(* Logix 5000 project; controller reports 1756-L63 rev 20.11; software revision 20.04; part 22 of 52 *)

        [1402].log_data[6].valid := 1, [1402].log_data[7].valid := 1, [1402].log_data[8].valid := 1, [1402].log_data[9].valid := 1, [1402].log_data[10].valid := 1, [1402].log_data[11].valid := 1, [1402].log_data[12].valid := 1, [1402].log_data[13].valid := 1, [1402].log_data[14].valid := 1, [1402].log_data[15].valid := 1, [1402].log_data[16].valid := 1, [1402].log_data[17].valid := 1, [1402].log_data[18].valid := 1, [1402].log_data[19].valid := 1, [1402].time.Year := 2023, [1402].time.Month := 1, [1402].time.Day := 14, [1402].time.Hour := 13, [1402].time.Minute := 14, [1402].time.Second := 59, [1403].log_data[0].min := 1.0, [1403].log_data[0].max := 1.0, [1403].log_data[0].total := 300.0, [1403].log_data[0].time := 300.0, [1403].log_data[0].minminute := 15, [1403].log_data[0].maxminute := 15, [1403].log_data[0].valid := 1, [1403].log_data[1].valid := 1, [1403].log_data[2].valid := 1, [1403].log_data[3].valid := 1, [1403].log_data[4].valid := 1, [1403].log_data[5].valid := 1, [1403].log_data[6].valid := 1, [1403].log_data[7].valid := 1, [1403].log_data[8].valid := 1, [1403].log_data[9].valid := 1, [1403].log_data[10].valid := 1, [1403].log_data[11].valid := 1, [1403].log_data[12].valid := 1, [1403].log_data[13].valid := 1, [1403].log_data[14].valid := 1, [1403].log_data[15].valid := 1, [1403].log_data[16].valid := 1, [1403].log_data[17].valid := 1, [1403].log_data[18].valid := 1, [1403].log_data[19].valid := 1, [1403].time.Year := 2023, [1403].time.Month := 1, [1403].time.Day := 14, [1403].time.Hour := 13, [1403].time.Minute := 19, [1403].time.Second := 59, [1404].log_data[0].min := 1.0, [1404].log_data[0].max := 1.0, [1404].log_data[0].total := 300.0, [1404].log_data[0].time := 300.0, [1404].log_data[0].minminute := 20, [1404].log_data[0].maxminute := 20, [1404].log_data[0].valid := 1, [1404].log_data[1].valid := 1,
        [1404].log_data[2].valid := 1, [1404].log_data[3].valid := 1, [1404].log_data[4].valid := 1, [1404].log_data[5].valid := 1, [1404].log_data[6].valid := 1, [1404].log_data[7].valid := 1, [1404].log_data[8].valid := 1, [1404].log_data[9].valid := 1, [1404].log_data[10].valid := 1, [1404].log_data[11].valid := 1, [1404].log_data[12].valid := 1, [1404].log_data[13].valid := 1, [1404].log_data[14].valid := 1, [1404].log_data[15].valid := 1, [1404].log_data[16].valid := 1, [1404].log_data[17].valid := 1, [1404].log_data[18].valid := 1, [1404].log_data[19].valid := 1, [1404].time.Year := 2023, [1404].time.Month := 1, [1404].time.Day := 14, [1404].time.Hour := 13, [1404].time.Minute := 24, [1404].time.Second := 59, [1405].log_data[0].min := 1.0, [1405].log_data[0].max := 1.0, [1405].log_data[0].total := 300.0, [1405].log_data[0].time := 300.0, [1405].log_data[0].minminute := 25, [1405].log_data[0].maxminute := 25, [1405].log_data[0].valid := 1, [1405].log_data[1].valid := 1, [1405].log_data[2].valid := 1, [1405].log_data[3].valid := 1, [1405].log_data[4].valid := 1, [1405].log_data[5].valid := 1, [1405].log_data[6].valid := 1, [1405].log_data[7].valid := 1, [1405].log_data[8].valid := 1, [1405].log_data[9].valid := 1, [1405].log_data[10].valid := 1, [1405].log_data[11].valid := 1, [1405].log_data[12].valid := 1, [1405].log_data[13].valid := 1, [1405].log_data[14].valid := 1, [1405].log_data[15].valid := 1, [1405].log_data[16].valid := 1, [1405].log_data[17].valid := 1, [1405].log_data[18].valid := 1, [1405].log_data[19].valid := 1, [1405].time.Year := 2023, [1405].time.Month := 1, [1405].time.Day := 14, [1405].time.Hour := 13, [1405].time.Minute := 29, [1405].time.Second := 59, [1406].log_data[0].min := 1.0, [1406].log_data[0].max := 1.0, [1406].log_data[0].total := 300.0, [1406].log_data[0].time := 300.0,
        [1406].log_data[0].minminute := 30, [1406].log_data[0].maxminute := 30, [1406].log_data[0].valid := 1, [1406].log_data[1].valid := 1, [1406].log_data[2].valid := 1, [1406].log_data[3].valid := 1, [1406].log_data[4].valid := 1, [1406].log_data[5].valid := 1, [1406].log_data[6].valid := 1, [1406].log_data[7].valid := 1, [1406].log_data[8].valid := 1, [1406].log_data[9].valid := 1, [1406].log_data[10].valid := 1, [1406].log_data[11].valid := 1, [1406].log_data[12].valid := 1, [1406].log_data[13].valid := 1, [1406].log_data[14].valid := 1, [1406].log_data[15].valid := 1, [1406].log_data[16].valid := 1, [1406].log_data[17].valid := 1, [1406].log_data[18].valid := 1, [1406].log_data[19].valid := 1, [1406].time.Year := 2023, [1406].time.Month := 1, [1406].time.Day := 14, [1406].time.Hour := 13, [1406].time.Minute := 34, [1406].time.Second := 59, [1407].log_data[0].min := 1.0, [1407].log_data[0].max := 1.0, [1407].log_data[0].total := 300.0, [1407].log_data[0].time := 300.0, [1407].log_data[0].minminute := 35, [1407].log_data[0].maxminute := 35, [1407].log_data[0].valid := 1, [1407].log_data[1].valid := 1, [1407].log_data[2].valid := 1, [1407].log_data[3].valid := 1, [1407].log_data[4].valid := 1, [1407].log_data[5].valid := 1, [1407].log_data[6].valid := 1, [1407].log_data[7].valid := 1, [1407].log_data[8].valid := 1, [1407].log_data[9].valid := 1, [1407].log_data[10].valid := 1, [1407].log_data[11].valid := 1, [1407].log_data[12].valid := 1, [1407].log_data[13].valid := 1, [1407].log_data[14].valid := 1, [1407].log_data[15].valid := 1, [1407].log_data[16].valid := 1, [1407].log_data[17].valid := 1, [1407].log_data[18].valid := 1, [1407].log_data[19].valid := 1, [1407].time.Year := 2023, [1407].time.Month := 1, [1407].time.Day := 14, [1407].time.Hour := 13, [1407].time.Minute := 39, [1407].time.Second := 59,
        [1408].log_data[0].min := 1.0, [1408].log_data[0].max := 1.0, [1408].log_data[0].total := 300.0, [1408].log_data[0].time := 300.0, [1408].log_data[0].minminute := 40, [1408].log_data[0].maxminute := 40, [1408].log_data[0].valid := 1, [1408].log_data[1].valid := 1, [1408].log_data[2].valid := 1, [1408].log_data[3].valid := 1, [1408].log_data[4].valid := 1, [1408].log_data[5].valid := 1, [1408].log_data[6].valid := 1, [1408].log_data[7].valid := 1, [1408].log_data[8].valid := 1, [1408].log_data[9].valid := 1, [1408].log_data[10].valid := 1, [1408].log_data[11].valid := 1, [1408].log_data[12].valid := 1, [1408].log_data[13].valid := 1, [1408].log_data[14].valid := 1, [1408].log_data[15].valid := 1, [1408].log_data[16].valid := 1, [1408].log_data[17].valid := 1, [1408].log_data[18].valid := 1, [1408].log_data[19].valid := 1, [1408].time.Year := 2023, [1408].time.Month := 1, [1408].time.Day := 14, [1408].time.Hour := 13, [1408].time.Minute := 44, [1408].time.Second := 59, [1409].log_data[0].min := 1.0, [1409].log_data[0].max := 1.0, [1409].log_data[0].total := 300.0, [1409].log_data[0].time := 300.0, [1409].log_data[0].minminute := 45, [1409].log_data[0].maxminute := 45, [1409].log_data[0].valid := 1, [1409].log_data[1].valid := 1, [1409].log_data[2].valid := 1, [1409].log_data[3].valid := 1, [1409].log_data[4].valid := 1, [1409].log_data[5].valid := 1, [1409].log_data[6].valid := 1, [1409].log_data[7].valid := 1, [1409].log_data[8].valid := 1, [1409].log_data[9].valid := 1, [1409].log_data[10].valid := 1, [1409].log_data[11].valid := 1, [1409].log_data[12].valid := 1, [1409].log_data[13].valid := 1, [1409].log_data[14].valid := 1, [1409].log_data[15].valid := 1, [1409].log_data[16].valid := 1, [1409].log_data[17].valid := 1, [1409].log_data[18].valid := 1, [1409].log_data[19].valid := 1, [1409].time.Year := 2023, [1409].time.Month := 1,
        [1409].time.Day := 14, [1409].time.Hour := 13, [1409].time.Minute := 49, [1409].time.Second := 59, [1410].log_data[0].min := 1.0, [1410].log_data[0].max := 1.0, [1410].log_data[0].total := 300.0, [1410].log_data[0].time := 300.0, [1410].log_data[0].minminute := 50, [1410].log_data[0].maxminute := 50, [1410].log_data[0].valid := 1, [1410].log_data[1].valid := 1, [1410].log_data[2].valid := 1, [1410].log_data[3].valid := 1, [1410].log_data[4].valid := 1, [1410].log_data[5].valid := 1, [1410].log_data[6].valid := 1, [1410].log_data[7].valid := 1, [1410].log_data[8].valid := 1, [1410].log_data[9].valid := 1, [1410].log_data[10].valid := 1, [1410].log_data[11].valid := 1, [1410].log_data[12].valid := 1, [1410].log_data[13].valid := 1, [1410].log_data[14].valid := 1, [1410].log_data[15].valid := 1, [1410].log_data[16].valid := 1, [1410].log_data[17].valid := 1, [1410].log_data[18].valid := 1, [1410].log_data[19].valid := 1, [1410].time.Year := 2023, [1410].time.Month := 1, [1410].time.Day := 14, [1410].time.Hour := 13, [1410].time.Minute := 54, [1410].time.Second := 59, [1411].log_data[0].min := 1.0, [1411].log_data[0].max := 1.0, [1411].log_data[0].total := 300.0, [1411].log_data[0].time := 300.0, [1411].log_data[0].minminute := 55, [1411].log_data[0].maxminute := 55, [1411].log_data[0].valid := 1, [1411].log_data[1].valid := 1, [1411].log_data[2].valid := 1, [1411].log_data[3].valid := 1, [1411].log_data[4].valid := 1, [1411].log_data[5].valid := 1, [1411].log_data[6].valid := 1, [1411].log_data[7].valid := 1, [1411].log_data[8].valid := 1, [1411].log_data[9].valid := 1, [1411].log_data[10].valid := 1, [1411].log_data[11].valid := 1, [1411].log_data[12].valid := 1, [1411].log_data[13].valid := 1, [1411].log_data[14].valid := 1, [1411].log_data[15].valid := 1, [1411].log_data[16].valid := 1, [1411].log_data[17].valid := 1,
        [1411].log_data[18].valid := 1, [1411].log_data[19].valid := 1, [1411].time.Year := 2023, [1411].time.Month := 1, [1411].time.Day := 14, [1411].time.Hour := 13, [1411].time.Minute := 59, [1411].time.Second := 59, [1412].log_data[0].min := 1.0, [1412].log_data[0].max := 1.0, [1412].log_data[0].total := 300.0, [1412].log_data[0].time := 300.0, [1412].log_data[0].valid := 1, [1412].log_data[1].valid := 1, [1412].log_data[2].valid := 1, [1412].log_data[3].valid := 1, [1412].log_data[4].valid := 1, [1412].log_data[5].valid := 1, [1412].log_data[6].valid := 1, [1412].log_data[7].valid := 1, [1412].log_data[8].valid := 1, [1412].log_data[9].valid := 1, [1412].log_data[10].valid := 1, [1412].log_data[11].valid := 1, [1412].log_data[12].valid := 1, [1412].log_data[13].valid := 1, [1412].log_data[14].valid := 1, [1412].log_data[15].valid := 1, [1412].log_data[16].valid := 1, [1412].log_data[17].valid := 1, [1412].log_data[18].valid := 1, [1412].log_data[19].valid := 1, [1412].time.Year := 2023, [1412].time.Month := 1, [1412].time.Day := 14, [1412].time.Hour := 14, [1412].time.Minute := 4, [1412].time.Second := 59, [1413].log_data[0].min := 1.0, [1413].log_data[0].max := 1.0, [1413].log_data[0].total := 300.0, [1413].log_data[0].time := 300.0, [1413].log_data[0].minminute := 5, [1413].log_data[0].maxminute := 5, [1413].log_data[0].valid := 1, [1413].log_data[1].valid := 1, [1413].log_data[2].valid := 1, [1413].log_data[3].valid := 1, [1413].log_data[4].valid := 1, [1413].log_data[5].valid := 1, [1413].log_data[6].valid := 1, [1413].log_data[7].valid := 1, [1413].log_data[8].valid := 1, [1413].log_data[9].valid := 1, [1413].log_data[10].valid := 1, [1413].log_data[11].valid := 1, [1413].log_data[12].valid := 1, [1413].log_data[13].valid := 1, [1413].log_data[14].valid := 1, [1413].log_data[15].valid := 1,
        [1413].log_data[16].valid := 1, [1413].log_data[17].valid := 1, [1413].log_data[18].valid := 1, [1413].log_data[19].valid := 1, [1413].time.Year := 2023, [1413].time.Month := 1, [1413].time.Day := 14, [1413].time.Hour := 14, [1413].time.Minute := 9, [1413].time.Second := 59, [1414].log_data[0].min := 1.0, [1414].log_data[0].max := 1.0, [1414].log_data[0].total := 300.0, [1414].log_data[0].time := 300.0, [1414].log_data[0].minminute := 10, [1414].log_data[0].maxminute := 10, [1414].log_data[0].valid := 1, [1414].log_data[1].valid := 1, [1414].log_data[2].valid := 1, [1414].log_data[3].valid := 1, [1414].log_data[4].valid := 1, [1414].log_data[5].valid := 1, [1414].log_data[6].valid := 1, [1414].log_data[7].valid := 1, [1414].log_data[8].valid := 1, [1414].log_data[9].valid := 1, [1414].log_data[10].valid := 1, [1414].log_data[11].valid := 1, [1414].log_data[12].valid := 1, [1414].log_data[13].valid := 1, [1414].log_data[14].valid := 1, [1414].log_data[15].valid := 1, [1414].log_data[16].valid := 1, [1414].log_data[17].valid := 1, [1414].log_data[18].valid := 1, [1414].log_data[19].valid := 1, [1414].time.Year := 2023, [1414].time.Month := 1, [1414].time.Day := 14, [1414].time.Hour := 14, [1414].time.Minute := 14, [1414].time.Second := 59, [1415].log_data[0].min := 1.0, [1415].log_data[0].max := 1.0, [1415].log_data[0].total := 300.0, [1415].log_data[0].time := 300.0, [1415].log_data[0].minminute := 15, [1415].log_data[0].maxminute := 15, [1415].log_data[0].valid := 1, [1415].log_data[1].valid := 1, [1415].log_data[2].valid := 1, [1415].log_data[3].valid := 1, [1415].log_data[4].valid := 1, [1415].log_data[5].valid := 1, [1415].log_data[6].valid := 1, [1415].log_data[7].valid := 1, [1415].log_data[8].valid := 1, [1415].log_data[9].valid := 1, [1415].log_data[10].valid := 1, [1415].log_data[11].valid := 1,
        [1415].log_data[12].valid := 1, [1415].log_data[13].valid := 1, [1415].log_data[14].valid := 1, [1415].log_data[15].valid := 1, [1415].log_data[16].valid := 1, [1415].log_data[17].valid := 1, [1415].log_data[18].valid := 1, [1415].log_data[19].valid := 1, [1415].time.Year := 2023, [1415].time.Month := 1, [1415].time.Day := 14, [1415].time.Hour := 14, [1415].time.Minute := 19, [1415].time.Second := 59, [1416].log_data[0].min := 1.0, [1416].log_data[0].max := 1.0, [1416].log_data[0].total := 300.0, [1416].log_data[0].time := 300.0, [1416].log_data[0].minminute := 20, [1416].log_data[0].maxminute := 20, [1416].log_data[0].valid := 1, [1416].log_data[1].valid := 1, [1416].log_data[2].valid := 1, [1416].log_data[3].valid := 1, [1416].log_data[4].valid := 1, [1416].log_data[5].valid := 1, [1416].log_data[6].valid := 1, [1416].log_data[7].valid := 1, [1416].log_data[8].valid := 1, [1416].log_data[9].valid := 1, [1416].log_data[10].valid := 1, [1416].log_data[11].valid := 1, [1416].log_data[12].valid := 1, [1416].log_data[13].valid := 1, [1416].log_data[14].valid := 1, [1416].log_data[15].valid := 1, [1416].log_data[16].valid := 1, [1416].log_data[17].valid := 1, [1416].log_data[18].valid := 1, [1416].log_data[19].valid := 1, [1416].time.Year := 2023, [1416].time.Month := 1, [1416].time.Day := 14, [1416].time.Hour := 14, [1416].time.Minute := 24, [1416].time.Second := 59, [1417].log_data[0].min := 1.0, [1417].log_data[0].max := 1.0, [1417].log_data[0].total := 300.0, [1417].log_data[0].time := 300.0, [1417].log_data[0].minminute := 25, [1417].log_data[0].maxminute := 25, [1417].log_data[0].valid := 1, [1417].log_data[1].valid := 1, [1417].log_data[2].valid := 1, [1417].log_data[3].valid := 1, [1417].log_data[4].valid := 1, [1417].log_data[5].valid := 1, [1417].log_data[6].valid := 1, [1417].log_data[7].valid := 1,
        [1417].log_data[8].valid := 1, [1417].log_data[9].valid := 1, [1417].log_data[10].valid := 1, [1417].log_data[11].valid := 1, [1417].log_data[12].valid := 1, [1417].log_data[13].valid := 1, [1417].log_data[14].valid := 1, [1417].log_data[15].valid := 1, [1417].log_data[16].valid := 1, [1417].log_data[17].valid := 1, [1417].log_data[18].valid := 1, [1417].log_data[19].valid := 1, [1417].time.Year := 2023, [1417].time.Month := 1, [1417].time.Day := 14, [1417].time.Hour := 14, [1417].time.Minute := 29, [1417].time.Second := 59, [1418].log_data[0].min := 1.0, [1418].log_data[0].max := 1.0, [1418].log_data[0].total := 300.0, [1418].log_data[0].time := 300.0, [1418].log_data[0].minminute := 30, [1418].log_data[0].maxminute := 30, [1418].log_data[0].valid := 1, [1418].log_data[1].valid := 1, [1418].log_data[2].valid := 1, [1418].log_data[3].valid := 1, [1418].log_data[4].valid := 1, [1418].log_data[5].valid := 1, [1418].log_data[6].valid := 1, [1418].log_data[7].valid := 1, [1418].log_data[8].valid := 1, [1418].log_data[9].valid := 1, [1418].log_data[10].valid := 1, [1418].log_data[11].valid := 1, [1418].log_data[12].valid := 1, [1418].log_data[13].valid := 1, [1418].log_data[14].valid := 1, [1418].log_data[15].valid := 1, [1418].log_data[16].valid := 1, [1418].log_data[17].valid := 1, [1418].log_data[18].valid := 1, [1418].log_data[19].valid := 1, [1418].time.Year := 2023, [1418].time.Month := 1, [1418].time.Day := 14, [1418].time.Hour := 14, [1418].time.Minute := 34, [1418].time.Second := 59, [1419].log_data[0].min := 1.0, [1419].log_data[0].max := 1.0, [1419].log_data[0].total := 300.0, [1419].log_data[0].time := 300.0, [1419].log_data[0].minminute := 35, [1419].log_data[0].maxminute := 35, [1419].log_data[0].valid := 1, [1419].log_data[1].valid := 1, [1419].log_data[2].valid := 1, [1419].log_data[3].valid := 1,
        [1419].log_data[4].valid := 1, [1419].log_data[5].valid := 1, [1419].log_data[6].valid := 1, [1419].log_data[7].valid := 1, [1419].log_data[8].valid := 1, [1419].log_data[9].valid := 1, [1419].log_data[10].valid := 1, [1419].log_data[11].valid := 1, [1419].log_data[12].valid := 1, [1419].log_data[13].valid := 1, [1419].log_data[14].valid := 1, [1419].log_data[15].valid := 1, [1419].log_data[16].valid := 1, [1419].log_data[17].valid := 1, [1419].log_data[18].valid := 1, [1419].log_data[19].valid := 1, [1419].time.Year := 2023, [1419].time.Month := 1, [1419].time.Day := 14, [1419].time.Hour := 14, [1419].time.Minute := 39, [1419].time.Second := 59, [1420].log_data[0].min := 1.0, [1420].log_data[0].max := 1.0, [1420].log_data[0].total := 300.0, [1420].log_data[0].time := 300.0, [1420].log_data[0].minminute := 40, [1420].log_data[0].maxminute := 40, [1420].log_data[0].valid := 1, [1420].log_data[1].valid := 1, [1420].log_data[2].valid := 1, [1420].log_data[3].valid := 1, [1420].log_data[4].valid := 1, [1420].log_data[5].valid := 1, [1420].log_data[6].valid := 1, [1420].log_data[7].valid := 1, [1420].log_data[8].valid := 1, [1420].log_data[9].valid := 1, [1420].log_data[10].valid := 1, [1420].log_data[11].valid := 1, [1420].log_data[12].valid := 1, [1420].log_data[13].valid := 1, [1420].log_data[14].valid := 1, [1420].log_data[15].valid := 1, [1420].log_data[16].valid := 1, [1420].log_data[17].valid := 1, [1420].log_data[18].valid := 1, [1420].log_data[19].valid := 1, [1420].time.Year := 2023, [1420].time.Month := 1, [1420].time.Day := 14, [1420].time.Hour := 14, [1420].time.Minute := 44, [1420].time.Second := 59, [1421].log_data[0].min := 1.0, [1421].log_data[0].max := 1.0, [1421].log_data[0].total := 300.0, [1421].log_data[0].time := 300.0, [1421].log_data[0].minminute := 45, [1421].log_data[0].maxminute := 45,
        [1421].log_data[0].valid := 1, [1421].log_data[1].valid := 1, [1421].log_data[2].valid := 1, [1421].log_data[3].valid := 1, [1421].log_data[4].valid := 1, [1421].log_data[5].valid := 1, [1421].log_data[6].valid := 1, [1421].log_data[7].valid := 1, [1421].log_data[8].valid := 1, [1421].log_data[9].valid := 1, [1421].log_data[10].valid := 1, [1421].log_data[11].valid := 1, [1421].log_data[12].valid := 1, [1421].log_data[13].valid := 1, [1421].log_data[14].valid := 1, [1421].log_data[15].valid := 1, [1421].log_data[16].valid := 1, [1421].log_data[17].valid := 1, [1421].log_data[18].valid := 1, [1421].log_data[19].valid := 1, [1421].time.Year := 2023, [1421].time.Month := 1, [1421].time.Day := 14, [1421].time.Hour := 14, [1421].time.Minute := 49, [1421].time.Second := 59, [1422].log_data[0].min := 1.0, [1422].log_data[0].max := 1.0, [1422].log_data[0].total := 300.0, [1422].log_data[0].time := 300.0, [1422].log_data[0].minminute := 50, [1422].log_data[0].maxminute := 50, [1422].log_data[0].valid := 1, [1422].log_data[1].valid := 1, [1422].log_data[2].valid := 1, [1422].log_data[3].valid := 1, [1422].log_data[4].valid := 1, [1422].log_data[5].valid := 1, [1422].log_data[6].valid := 1, [1422].log_data[7].valid := 1, [1422].log_data[8].valid := 1, [1422].log_data[9].valid := 1, [1422].log_data[10].valid := 1, [1422].log_data[11].valid := 1, [1422].log_data[12].valid := 1, [1422].log_data[13].valid := 1, [1422].log_data[14].valid := 1, [1422].log_data[15].valid := 1, [1422].log_data[16].valid := 1, [1422].log_data[17].valid := 1, [1422].log_data[18].valid := 1, [1422].log_data[19].valid := 1, [1422].time.Year := 2023, [1422].time.Month := 1, [1422].time.Day := 14, [1422].time.Hour := 14, [1422].time.Minute := 54, [1422].time.Second := 59, [1423].log_data[0].min := 1.0, [1423].log_data[0].max := 1.0,
        [1423].log_data[0].total := 300.0, [1423].log_data[0].time := 300.0, [1423].log_data[0].minminute := 55, [1423].log_data[0].maxminute := 55, [1423].log_data[0].valid := 1, [1423].log_data[1].valid := 1, [1423].log_data[2].valid := 1, [1423].log_data[3].valid := 1, [1423].log_data[4].valid := 1, [1423].log_data[5].valid := 1, [1423].log_data[6].valid := 1, [1423].log_data[7].valid := 1, [1423].log_data[8].valid := 1, [1423].log_data[9].valid := 1, [1423].log_data[10].valid := 1, [1423].log_data[11].valid := 1, [1423].log_data[12].valid := 1, [1423].log_data[13].valid := 1, [1423].log_data[14].valid := 1, [1423].log_data[15].valid := 1, [1423].log_data[16].valid := 1, [1423].log_data[17].valid := 1, [1423].log_data[18].valid := 1, [1423].log_data[19].valid := 1, [1423].time.Year := 2023, [1423].time.Month := 1, [1423].time.Day := 14, [1423].time.Hour := 14, [1423].time.Minute := 59, [1423].time.Second := 59, [1424].log_data[0].min := 1.0, [1424].log_data[0].max := 1.0, [1424].log_data[0].total := 300.0, [1424].log_data[0].time := 300.0, [1424].log_data[0].valid := 1, [1424].log_data[1].valid := 1, [1424].log_data[2].valid := 1, [1424].log_data[3].valid := 1, [1424].log_data[4].valid := 1, [1424].log_data[5].valid := 1, [1424].log_data[6].valid := 1, [1424].log_data[7].valid := 1, [1424].log_data[8].valid := 1, [1424].log_data[9].valid := 1, [1424].log_data[10].valid := 1, [1424].log_data[11].valid := 1, [1424].log_data[12].valid := 1, [1424].log_data[13].valid := 1, [1424].log_data[14].valid := 1, [1424].log_data[15].valid := 1, [1424].log_data[16].valid := 1, [1424].log_data[17].valid := 1, [1424].log_data[18].valid := 1, [1424].log_data[19].valid := 1, [1424].time.Year := 2023, [1424].time.Month := 1, [1424].time.Day := 14, [1424].time.Hour := 15, [1424].time.Minute := 4, [1424].time.Second := 59,
        [1425].log_data[0].min := 1.0, [1425].log_data[0].max := 1.0, [1425].log_data[0].total := 300.0, [1425].log_data[0].time := 300.0, [1425].log_data[0].minminute := 5, [1425].log_data[0].maxminute := 5, [1425].log_data[0].valid := 1, [1425].log_data[1].valid := 1, [1425].log_data[2].valid := 1, [1425].log_data[3].valid := 1, [1425].log_data[4].valid := 1, [1425].log_data[5].valid := 1, [1425].log_data[6].valid := 1, [1425].log_data[7].valid := 1, [1425].log_data[8].valid := 1, [1425].log_data[9].valid := 1, [1425].log_data[10].valid := 1, [1425].log_data[11].valid := 1, [1425].log_data[12].valid := 1, [1425].log_data[13].valid := 1, [1425].log_data[14].valid := 1, [1425].log_data[15].valid := 1, [1425].log_data[16].valid := 1, [1425].log_data[17].valid := 1, [1425].log_data[18].valid := 1, [1425].log_data[19].valid := 1, [1425].time.Year := 2023, [1425].time.Month := 1, [1425].time.Day := 14, [1425].time.Hour := 15, [1425].time.Minute := 9, [1425].time.Second := 59, [1426].log_data[0].min := 1.0, [1426].log_data[0].max := 1.0, [1426].log_data[0].total := 300.0, [1426].log_data[0].time := 300.0, [1426].log_data[0].minminute := 10, [1426].log_data[0].maxminute := 10, [1426].log_data[0].valid := 1, [1426].log_data[1].valid := 1, [1426].log_data[2].valid := 1, [1426].log_data[3].valid := 1, [1426].log_data[4].valid := 1, [1426].log_data[5].valid := 1, [1426].log_data[6].valid := 1, [1426].log_data[7].valid := 1, [1426].log_data[8].valid := 1, [1426].log_data[9].valid := 1, [1426].log_data[10].valid := 1, [1426].log_data[11].valid := 1, [1426].log_data[12].valid := 1, [1426].log_data[13].valid := 1, [1426].log_data[14].valid := 1, [1426].log_data[15].valid := 1, [1426].log_data[16].valid := 1, [1426].log_data[17].valid := 1, [1426].log_data[18].valid := 1, [1426].log_data[19].valid := 1, [1426].time.Year := 2023, [1426].time.Month := 1,
        [1426].time.Day := 14, [1426].time.Hour := 15, [1426].time.Minute := 14, [1426].time.Second := 59, [1427].log_data[0].min := 1.0, [1427].log_data[0].max := 1.0, [1427].log_data[0].total := 300.0, [1427].log_data[0].time := 300.0, [1427].log_data[0].minminute := 15, [1427].log_data[0].maxminute := 15, [1427].log_data[0].valid := 1, [1427].log_data[1].valid := 1, [1427].log_data[2].valid := 1, [1427].log_data[3].valid := 1, [1427].log_data[4].valid := 1, [1427].log_data[5].valid := 1, [1427].log_data[6].valid := 1, [1427].log_data[7].valid := 1, [1427].log_data[8].valid := 1, [1427].log_data[9].valid := 1, [1427].log_data[10].valid := 1, [1427].log_data[11].valid := 1, [1427].log_data[12].valid := 1, [1427].log_data[13].valid := 1, [1427].log_data[14].valid := 1, [1427].log_data[15].valid := 1, [1427].log_data[16].valid := 1, [1427].log_data[17].valid := 1, [1427].log_data[18].valid := 1, [1427].log_data[19].valid := 1, [1427].time.Year := 2023, [1427].time.Month := 1, [1427].time.Day := 14, [1427].time.Hour := 15, [1427].time.Minute := 19, [1427].time.Second := 59, [1428].log_data[0].min := 1.0, [1428].log_data[0].max := 1.0, [1428].log_data[0].total := 300.0, [1428].log_data[0].time := 300.0, [1428].log_data[0].minminute := 20, [1428].log_data[0].maxminute := 20, [1428].log_data[0].valid := 1, [1428].log_data[1].valid := 1, [1428].log_data[2].valid := 1, [1428].log_data[3].valid := 1, [1428].log_data[4].valid := 1, [1428].log_data[5].valid := 1, [1428].log_data[6].valid := 1, [1428].log_data[7].valid := 1, [1428].log_data[8].valid := 1, [1428].log_data[9].valid := 1, [1428].log_data[10].valid := 1, [1428].log_data[11].valid := 1, [1428].log_data[12].valid := 1, [1428].log_data[13].valid := 1, [1428].log_data[14].valid := 1, [1428].log_data[15].valid := 1, [1428].log_data[16].valid := 1, [1428].log_data[17].valid := 1,
        [1428].log_data[18].valid := 1, [1428].log_data[19].valid := 1, [1428].time.Year := 2023, [1428].time.Month := 1, [1428].time.Day := 14, [1428].time.Hour := 15, [1428].time.Minute := 24, [1428].time.Second := 59, [1429].log_data[0].min := 1.0, [1429].log_data[0].max := 1.0, [1429].log_data[0].total := 300.0, [1429].log_data[0].time := 300.0, [1429].log_data[0].minminute := 25, [1429].log_data[0].maxminute := 25, [1429].log_data[0].valid := 1, [1429].log_data[1].valid := 1, [1429].log_data[2].valid := 1, [1429].log_data[3].valid := 1, [1429].log_data[4].valid := 1, [1429].log_data[5].valid := 1, [1429].log_data[6].valid := 1, [1429].log_data[7].valid := 1, [1429].log_data[8].valid := 1, [1429].log_data[9].valid := 1, [1429].log_data[10].valid := 1, [1429].log_data[11].valid := 1, [1429].log_data[12].valid := 1, [1429].log_data[13].valid := 1, [1429].log_data[14].valid := 1, [1429].log_data[15].valid := 1, [1429].log_data[16].valid := 1, [1429].log_data[17].valid := 1, [1429].log_data[18].valid := 1, [1429].log_data[19].valid := 1, [1429].time.Year := 2023, [1429].time.Month := 1, [1429].time.Day := 14, [1429].time.Hour := 15, [1429].time.Minute := 29, [1429].time.Second := 59, [1430].log_data[0].min := 1.0, [1430].log_data[0].max := 1.0, [1430].log_data[0].total := 300.0, [1430].log_data[0].time := 300.0, [1430].log_data[0].minminute := 30, [1430].log_data[0].maxminute := 30, [1430].log_data[0].valid := 1, [1430].log_data[1].valid := 1, [1430].log_data[2].valid := 1, [1430].log_data[3].valid := 1, [1430].log_data[4].valid := 1, [1430].log_data[5].valid := 1, [1430].log_data[6].valid := 1, [1430].log_data[7].valid := 1, [1430].log_data[8].valid := 1, [1430].log_data[9].valid := 1, [1430].log_data[10].valid := 1, [1430].log_data[11].valid := 1, [1430].log_data[12].valid := 1, [1430].log_data[13].valid := 1,
        [1430].log_data[14].valid := 1, [1430].log_data[15].valid := 1, [1430].log_data[16].valid := 1, [1430].log_data[17].valid := 1, [1430].log_data[18].valid := 1, [1430].log_data[19].valid := 1, [1430].time.Year := 2023, [1430].time.Month := 1, [1430].time.Day := 14, [1430].time.Hour := 15, [1430].time.Minute := 34, [1430].time.Second := 59, [1431].log_data[0].min := 1.0, [1431].log_data[0].max := 1.0, [1431].log_data[0].total := 300.0, [1431].log_data[0].time := 300.0, [1431].log_data[0].minminute := 35, [1431].log_data[0].maxminute := 35, [1431].log_data[0].valid := 1, [1431].log_data[1].valid := 1, [1431].log_data[2].valid := 1, [1431].log_data[3].valid := 1, [1431].log_data[4].valid := 1, [1431].log_data[5].valid := 1, [1431].log_data[6].valid := 1, [1431].log_data[7].valid := 1, [1431].log_data[8].valid := 1, [1431].log_data[9].valid := 1, [1431].log_data[10].valid := 1, [1431].log_data[11].valid := 1, [1431].log_data[12].valid := 1, [1431].log_data[13].valid := 1, [1431].log_data[14].valid := 1, [1431].log_data[15].valid := 1, [1431].log_data[16].valid := 1, [1431].log_data[17].valid := 1, [1431].log_data[18].valid := 1, [1431].log_data[19].valid := 1, [1431].time.Year := 2023, [1431].time.Month := 1, [1431].time.Day := 14, [1431].time.Hour := 15, [1431].time.Minute := 39, [1431].time.Second := 59, [1432].log_data[0].min := 1.0, [1432].log_data[0].max := 1.0, [1432].log_data[0].total := 300.0, [1432].log_data[0].time := 300.0, [1432].log_data[0].minminute := 40, [1432].log_data[0].maxminute := 40, [1432].log_data[0].valid := 1, [1432].log_data[1].valid := 1, [1432].log_data[2].valid := 1, [1432].log_data[3].valid := 1, [1432].log_data[4].valid := 1, [1432].log_data[5].valid := 1, [1432].log_data[6].valid := 1, [1432].log_data[7].valid := 1, [1432].log_data[8].valid := 1, [1432].log_data[9].valid := 1,
        [1432].log_data[10].valid := 1, [1432].log_data[11].valid := 1, [1432].log_data[12].valid := 1, [1432].log_data[13].valid := 1, [1432].log_data[14].valid := 1, [1432].log_data[15].valid := 1, [1432].log_data[16].valid := 1, [1432].log_data[17].valid := 1, [1432].log_data[18].valid := 1, [1432].log_data[19].valid := 1, [1432].time.Year := 2023, [1432].time.Month := 1, [1432].time.Day := 14, [1432].time.Hour := 15, [1432].time.Minute := 44, [1432].time.Second := 59, [1433].log_data[0].min := 1.0, [1433].log_data[0].max := 1.0, [1433].log_data[0].total := 300.0, [1433].log_data[0].time := 300.0, [1433].log_data[0].minminute := 45, [1433].log_data[0].maxminute := 45, [1433].log_data[0].valid := 1, [1433].log_data[1].valid := 1, [1433].log_data[2].valid := 1, [1433].log_data[3].valid := 1, [1433].log_data[4].valid := 1, [1433].log_data[5].valid := 1, [1433].log_data[6].valid := 1, [1433].log_data[7].valid := 1, [1433].log_data[8].valid := 1, [1433].log_data[9].valid := 1, [1433].log_data[10].valid := 1, [1433].log_data[11].valid := 1, [1433].log_data[12].valid := 1, [1433].log_data[13].valid := 1, [1433].log_data[14].valid := 1, [1433].log_data[15].valid := 1, [1433].log_data[16].valid := 1, [1433].log_data[17].valid := 1, [1433].log_data[18].valid := 1, [1433].log_data[19].valid := 1, [1433].time.Year := 2023, [1433].time.Month := 1, [1433].time.Day := 14, [1433].time.Hour := 15, [1433].time.Minute := 49, [1433].time.Second := 59, [1434].log_data[0].min := 1.0, [1434].log_data[0].max := 1.0, [1434].log_data[0].total := 300.0, [1434].log_data[0].time := 300.0, [1434].log_data[0].minminute := 50, [1434].log_data[0].maxminute := 50, [1434].log_data[0].valid := 1, [1434].log_data[1].valid := 1, [1434].log_data[2].valid := 1, [1434].log_data[3].valid := 1, [1434].log_data[4].valid := 1, [1434].log_data[5].valid := 1,
        [1434].log_data[6].valid := 1, [1434].log_data[7].valid := 1, [1434].log_data[8].valid := 1, [1434].log_data[9].valid := 1, [1434].log_data[10].valid := 1, [1434].log_data[11].valid := 1, [1434].log_data[12].valid := 1, [1434].log_data[13].valid := 1, [1434].log_data[14].valid := 1, [1434].log_data[15].valid := 1, [1434].log_data[16].valid := 1, [1434].log_data[17].valid := 1, [1434].log_data[18].valid := 1, [1434].log_data[19].valid := 1, [1434].time.Year := 2023, [1434].time.Month := 1, [1434].time.Day := 14, [1434].time.Hour := 15, [1434].time.Minute := 54, [1434].time.Second := 59, [1435].log_data[0].min := 1.0, [1435].log_data[0].max := 1.0, [1435].log_data[0].total := 300.0, [1435].log_data[0].time := 300.0, [1435].log_data[0].minminute := 55, [1435].log_data[0].maxminute := 55, [1435].log_data[0].valid := 1, [1435].log_data[1].valid := 1, [1435].log_data[2].valid := 1, [1435].log_data[3].valid := 1, [1435].log_data[4].valid := 1, [1435].log_data[5].valid := 1, [1435].log_data[6].valid := 1, [1435].log_data[7].valid := 1, [1435].log_data[8].valid := 1, [1435].log_data[9].valid := 1, [1435].log_data[10].valid := 1, [1435].log_data[11].valid := 1, [1435].log_data[12].valid := 1, [1435].log_data[13].valid := 1, [1435].log_data[14].valid := 1, [1435].log_data[15].valid := 1, [1435].log_data[16].valid := 1, [1435].log_data[17].valid := 1, [1435].log_data[18].valid := 1, [1435].log_data[19].valid := 1, [1435].time.Year := 2023, [1435].time.Month := 1, [1435].time.Day := 14, [1435].time.Hour := 15, [1435].time.Minute := 59, [1435].time.Second := 59, [1436].log_data[0].min := 1.0, [1436].log_data[0].max := 1.0, [1436].log_data[0].total := 300.0, [1436].log_data[0].time := 300.0, [1436].log_data[0].valid := 1, [1436].log_data[1].valid := 1, [1436].log_data[2].valid := 1, [1436].log_data[3].valid := 1,
        [1436].log_data[4].valid := 1, [1436].log_data[5].valid := 1, [1436].log_data[6].valid := 1, [1436].log_data[7].valid := 1, [1436].log_data[8].valid := 1, [1436].log_data[9].valid := 1, [1436].log_data[10].valid := 1, [1436].log_data[11].valid := 1, [1436].log_data[12].valid := 1, [1436].log_data[13].valid := 1, [1436].log_data[14].valid := 1, [1436].log_data[15].valid := 1, [1436].log_data[16].valid := 1, [1436].log_data[17].valid := 1, [1436].log_data[18].valid := 1, [1436].log_data[19].valid := 1, [1436].time.Year := 2023, [1436].time.Month := 1, [1436].time.Day := 14, [1436].time.Hour := 16, [1436].time.Minute := 4, [1436].time.Second := 59, [1437].log_data[0].min := 1.0, [1437].log_data[0].max := 1.0, [1437].log_data[0].total := 300.0, [1437].log_data[0].time := 300.0, [1437].log_data[0].minminute := 5, [1437].log_data[0].maxminute := 5, [1437].log_data[0].valid := 1, [1437].log_data[1].valid := 1, [1437].log_data[2].valid := 1, [1437].log_data[3].valid := 1, [1437].log_data[4].valid := 1, [1437].log_data[5].valid := 1, [1437].log_data[6].valid := 1, [1437].log_data[7].valid := 1, [1437].log_data[8].valid := 1, [1437].log_data[9].valid := 1, [1437].log_data[10].valid := 1, [1437].log_data[11].valid := 1, [1437].log_data[12].valid := 1, [1437].log_data[13].valid := 1, [1437].log_data[14].valid := 1, [1437].log_data[15].valid := 1, [1437].log_data[16].valid := 1, [1437].log_data[17].valid := 1, [1437].log_data[18].valid := 1, [1437].log_data[19].valid := 1, [1437].time.Year := 2023, [1437].time.Month := 1, [1437].time.Day := 14, [1437].time.Hour := 16, [1437].time.Minute := 9, [1437].time.Second := 59, [1438].log_data[0].min := 1.0, [1438].log_data[0].max := 1.0, [1438].log_data[0].total := 300.0, [1438].log_data[0].time := 300.0, [1438].log_data[0].minminute := 10, [1438].log_data[0].maxminute := 10,
        [1438].log_data[0].valid := 1, [1438].log_data[1].valid := 1, [1438].log_data[2].valid := 1, [1438].log_data[3].valid := 1, [1438].log_data[4].valid := 1, [1438].log_data[5].valid := 1, [1438].log_data[6].valid := 1, [1438].log_data[7].valid := 1, [1438].log_data[8].valid := 1, [1438].log_data[9].valid := 1, [1438].log_data[10].valid := 1, [1438].log_data[11].valid := 1, [1438].log_data[12].valid := 1, [1438].log_data[13].valid := 1, [1438].log_data[14].valid := 1, [1438].log_data[15].valid := 1, [1438].log_data[16].valid := 1, [1438].log_data[17].valid := 1, [1438].log_data[18].valid := 1, [1438].log_data[19].valid := 1, [1438].time.Year := 2023, [1438].time.Month := 1, [1438].time.Day := 14, [1438].time.Hour := 16, [1438].time.Minute := 14, [1438].time.Second := 59, [1439].log_data[0].min := 1.0, [1439].log_data[0].max := 1.0, [1439].log_data[0].total := 300.0, [1439].log_data[0].time := 300.0, [1439].log_data[0].minminute := 15, [1439].log_data[0].maxminute := 15, [1439].log_data[0].valid := 1, [1439].log_data[1].valid := 1, [1439].log_data[2].valid := 1, [1439].log_data[3].valid := 1, [1439].log_data[4].valid := 1, [1439].log_data[5].valid := 1, [1439].log_data[6].valid := 1, [1439].log_data[7].valid := 1, [1439].log_data[8].valid := 1, [1439].log_data[9].valid := 1, [1439].log_data[10].valid := 1, [1439].log_data[11].valid := 1, [1439].log_data[12].valid := 1, [1439].log_data[13].valid := 1, [1439].log_data[14].valid := 1, [1439].log_data[15].valid := 1, [1439].log_data[16].valid := 1, [1439].log_data[17].valid := 1, [1439].log_data[18].valid := 1, [1439].log_data[19].valid := 1, [1439].time.Year := 2023, [1439].time.Month := 1, [1439].time.Day := 14, [1439].time.Hour := 16, [1439].time.Minute := 19, [1439].time.Second := 59, [1440].log_data[0].min := 1.0, [1440].log_data[0].max := 1.0,
        [1440].log_data[0].total := 300.0, [1440].log_data[0].time := 300.0, [1440].log_data[0].minminute := 20, [1440].log_data[0].maxminute := 20, [1440].log_data[0].valid := 1, [1440].log_data[1].valid := 1, [1440].log_data[2].valid := 1, [1440].log_data[3].valid := 1, [1440].log_data[4].valid := 1, [1440].log_data[5].valid := 1, [1440].log_data[6].valid := 1, [1440].log_data[7].valid := 1, [1440].log_data[8].valid := 1, [1440].log_data[9].valid := 1, [1440].log_data[10].valid := 1, [1440].log_data[11].valid := 1, [1440].log_data[12].valid := 1, [1440].log_data[13].valid := 1, [1440].log_data[14].valid := 1, [1440].log_data[15].valid := 1, [1440].log_data[16].valid := 1, [1440].log_data[17].valid := 1, [1440].log_data[18].valid := 1, [1440].log_data[19].valid := 1, [1440].time.Year := 2023, [1440].time.Month := 1, [1440].time.Day := 14, [1440].time.Hour := 16, [1440].time.Minute := 24, [1440].time.Second := 59, [1441].log_data[0].min := 1.0, [1441].log_data[0].max := 1.0, [1441].log_data[0].total := 300.0, [1441].log_data[0].time := 300.0, [1441].log_data[0].minminute := 25, [1441].log_data[0].maxminute := 25, [1441].log_data[0].valid := 1, [1441].log_data[1].valid := 1, [1441].log_data[2].valid := 1, [1441].log_data[3].valid := 1, [1441].log_data[4].valid := 1, [1441].log_data[5].valid := 1, [1441].log_data[6].valid := 1, [1441].log_data[7].valid := 1, [1441].log_data[8].valid := 1, [1441].log_data[9].valid := 1, [1441].log_data[10].valid := 1, [1441].log_data[11].valid := 1, [1441].log_data[12].valid := 1, [1441].log_data[13].valid := 1, [1441].log_data[14].valid := 1, [1441].log_data[15].valid := 1, [1441].log_data[16].valid := 1, [1441].log_data[17].valid := 1, [1441].log_data[18].valid := 1, [1441].log_data[19].valid := 1, [1441].time.Year := 2023, [1441].time.Month := 1, [1441].time.Day := 14, [1441].time.Hour := 16,
        [1441].time.Minute := 29, [1441].time.Second := 59, [1442].log_data[0].min := 1.0, [1442].log_data[0].max := 1.0, [1442].log_data[0].total := 300.0, [1442].log_data[0].time := 300.0, [1442].log_data[0].minminute := 30, [1442].log_data[0].maxminute := 30, [1442].log_data[0].valid := 1, [1442].log_data[1].valid := 1, [1442].log_data[2].valid := 1, [1442].log_data[3].valid := 1, [1442].log_data[4].valid := 1, [1442].log_data[5].valid := 1, [1442].log_data[6].valid := 1, [1442].log_data[7].valid := 1, [1442].log_data[8].valid := 1, [1442].log_data[9].valid := 1, [1442].log_data[10].valid := 1, [1442].log_data[11].valid := 1, [1442].log_data[12].valid := 1, [1442].log_data[13].valid := 1, [1442].log_data[14].valid := 1, [1442].log_data[15].valid := 1, [1442].log_data[16].valid := 1, [1442].log_data[17].valid := 1, [1442].log_data[18].valid := 1, [1442].log_data[19].valid := 1, [1442].time.Year := 2023, [1442].time.Month := 1, [1442].time.Day := 14, [1442].time.Hour := 16, [1442].time.Minute := 34, [1442].time.Second := 59, [1443].log_data[0].min := 1.0, [1443].log_data[0].max := 1.0, [1443].log_data[0].total := 300.0, [1443].log_data[0].time := 300.0, [1443].log_data[0].minminute := 35, [1443].log_data[0].maxminute := 35, [1443].log_data[0].valid := 1, [1443].log_data[1].valid := 1, [1443].log_data[2].valid := 1, [1443].log_data[3].valid := 1, [1443].log_data[4].valid := 1, [1443].log_data[5].valid := 1, [1443].log_data[6].valid := 1, [1443].log_data[7].valid := 1, [1443].log_data[8].valid := 1, [1443].log_data[9].valid := 1, [1443].log_data[10].valid := 1, [1443].log_data[11].valid := 1, [1443].log_data[12].valid := 1, [1443].log_data[13].valid := 1, [1443].log_data[14].valid := 1, [1443].log_data[15].valid := 1, [1443].log_data[16].valid := 1, [1443].log_data[17].valid := 1, [1443].log_data[18].valid := 1, [1443].log_data[19].valid := 1,
        [1443].time.Year := 2023, [1443].time.Month := 1, [1443].time.Day := 14, [1443].time.Hour := 16, [1443].time.Minute := 39, [1443].time.Second := 59, [1444].log_data[0].min := 1.0, [1444].log_data[0].max := 1.0, [1444].log_data[0].total := 300.0, [1444].log_data[0].time := 300.0, [1444].log_data[0].minminute := 40, [1444].log_data[0].maxminute := 40, [1444].log_data[0].valid := 1, [1444].log_data[1].valid := 1, [1444].log_data[2].valid := 1, [1444].log_data[3].valid := 1, [1444].log_data[4].valid := 1, [1444].log_data[5].valid := 1, [1444].log_data[6].valid := 1, [1444].log_data[7].valid := 1, [1444].log_data[8].valid := 1, [1444].log_data[9].valid := 1, [1444].log_data[10].valid := 1, [1444].log_data[11].valid := 1, [1444].log_data[12].valid := 1, [1444].log_data[13].valid := 1, [1444].log_data[14].valid := 1, [1444].log_data[15].valid := 1, [1444].log_data[16].valid := 1, [1444].log_data[17].valid := 1, [1444].log_data[18].valid := 1, [1444].log_data[19].valid := 1, [1444].time.Year := 2023, [1444].time.Month := 1, [1444].time.Day := 14, [1444].time.Hour := 16, [1444].time.Minute := 44, [1444].time.Second := 59, [1445].log_data[0].min := 1.0, [1445].log_data[0].max := 1.0, [1445].log_data[0].total := 300.0, [1445].log_data[0].time := 300.0, [1445].log_data[0].minminute := 45, [1445].log_data[0].maxminute := 45, [1445].log_data[0].valid := 1, [1445].log_data[1].valid := 1, [1445].log_data[2].valid := 1, [1445].log_data[3].valid := 1, [1445].log_data[4].valid := 1, [1445].log_data[5].valid := 1, [1445].log_data[6].valid := 1, [1445].log_data[7].valid := 1, [1445].log_data[8].valid := 1, [1445].log_data[9].valid := 1, [1445].log_data[10].valid := 1, [1445].log_data[11].valid := 1, [1445].log_data[12].valid := 1, [1445].log_data[13].valid := 1, [1445].log_data[14].valid := 1, [1445].log_data[15].valid := 1,
        [1445].log_data[16].valid := 1, [1445].log_data[17].valid := 1, [1445].log_data[18].valid := 1, [1445].log_data[19].valid := 1, [1445].time.Year := 2023, [1445].time.Month := 1, [1445].time.Day := 14, [1445].time.Hour := 16, [1445].time.Minute := 49, [1445].time.Second := 59, [1446].log_data[0].min := 1.0, [1446].log_data[0].max := 1.0, [1446].log_data[0].total := 300.0, [1446].log_data[0].time := 300.0, [1446].log_data[0].minminute := 50, [1446].log_data[0].maxminute := 50, [1446].log_data[0].valid := 1, [1446].log_data[1].valid := 1, [1446].log_data[2].valid := 1, [1446].log_data[3].valid := 1, [1446].log_data[4].valid := 1, [1446].log_data[5].valid := 1, [1446].log_data[6].valid := 1, [1446].log_data[7].valid := 1, [1446].log_data[8].valid := 1, [1446].log_data[9].valid := 1, [1446].log_data[10].valid := 1, [1446].log_data[11].valid := 1, [1446].log_data[12].valid := 1, [1446].log_data[13].valid := 1, [1446].log_data[14].valid := 1, [1446].log_data[15].valid := 1, [1446].log_data[16].valid := 1, [1446].log_data[17].valid := 1, [1446].log_data[18].valid := 1, [1446].log_data[19].valid := 1, [1446].time.Year := 2023, [1446].time.Month := 1, [1446].time.Day := 14, [1446].time.Hour := 16, [1446].time.Minute := 54, [1446].time.Second := 59, [1447].log_data[0].min := 1.0, [1447].log_data[0].max := 1.0, [1447].log_data[0].total := 300.0, [1447].log_data[0].time := 300.0, [1447].log_data[0].minminute := 55, [1447].log_data[0].maxminute := 55, [1447].log_data[0].valid := 1, [1447].log_data[1].valid := 1, [1447].log_data[2].valid := 1, [1447].log_data[3].valid := 1, [1447].log_data[4].valid := 1, [1447].log_data[5].valid := 1, [1447].log_data[6].valid := 1, [1447].log_data[7].valid := 1, [1447].log_data[8].valid := 1, [1447].log_data[9].valid := 1, [1447].log_data[10].valid := 1, [1447].log_data[11].valid := 1,
        [1447].log_data[12].valid := 1, [1447].log_data[13].valid := 1, [1447].log_data[14].valid := 1, [1447].log_data[15].valid := 1, [1447].log_data[16].valid := 1, [1447].log_data[17].valid := 1, [1447].log_data[18].valid := 1, [1447].log_data[19].valid := 1, [1447].time.Year := 2023, [1447].time.Month := 1, [1447].time.Day := 14, [1447].time.Hour := 16, [1447].time.Minute := 59, [1447].time.Second := 59, [1448].log_data[0].min := 1.0, [1448].log_data[0].max := 1.0, [1448].log_data[0].total := 300.0, [1448].log_data[0].time := 300.0, [1448].log_data[0].valid := 1, [1448].log_data[1].valid := 1, [1448].log_data[2].valid := 1, [1448].log_data[3].valid := 1, [1448].log_data[4].valid := 1, [1448].log_data[5].valid := 1, [1448].log_data[6].valid := 1, [1448].log_data[7].valid := 1, [1448].log_data[8].valid := 1, [1448].log_data[9].valid := 1, [1448].log_data[10].valid := 1, [1448].log_data[11].valid := 1, [1448].log_data[12].valid := 1, [1448].log_data[13].valid := 1, [1448].log_data[14].valid := 1, [1448].log_data[15].valid := 1, [1448].log_data[16].valid := 1, [1448].log_data[17].valid := 1, [1448].log_data[18].valid := 1, [1448].log_data[19].valid := 1, [1448].time.Year := 2023, [1448].time.Month := 1, [1448].time.Day := 14, [1448].time.Hour := 17, [1448].time.Minute := 4, [1448].time.Second := 59, [1449].log_data[0].min := 1.0, [1449].log_data[0].max := 1.0, [1449].log_data[0].total := 300.0, [1449].log_data[0].time := 300.0, [1449].log_data[0].minminute := 5, [1449].log_data[0].maxminute := 5, [1449].log_data[0].valid := 1, [1449].log_data[1].valid := 1, [1449].log_data[2].valid := 1, [1449].log_data[3].valid := 1, [1449].log_data[4].valid := 1, [1449].log_data[5].valid := 1, [1449].log_data[6].valid := 1, [1449].log_data[7].valid := 1, [1449].log_data[8].valid := 1, [1449].log_data[9].valid := 1,
        [1449].log_data[10].valid := 1, [1449].log_data[11].valid := 1, [1449].log_data[12].valid := 1, [1449].log_data[13].valid := 1, [1449].log_data[14].valid := 1, [1449].log_data[15].valid := 1, [1449].log_data[16].valid := 1, [1449].log_data[17].valid := 1, [1449].log_data[18].valid := 1, [1449].log_data[19].valid := 1, [1449].time.Year := 2023, [1449].time.Month := 1, [1449].time.Day := 14, [1449].time.Hour := 17, [1449].time.Minute := 9, [1449].time.Second := 59, [1450].log_data[0].min := 1.0, [1450].log_data[0].max := 1.0, [1450].log_data[0].total := 300.0, [1450].log_data[0].time := 300.0, [1450].log_data[0].minminute := 10, [1450].log_data[0].maxminute := 10, [1450].log_data[0].valid := 1, [1450].log_data[1].valid := 1, [1450].log_data[2].valid := 1, [1450].log_data[3].valid := 1, [1450].log_data[4].valid := 1, [1450].log_data[5].valid := 1, [1450].log_data[6].valid := 1, [1450].log_data[7].valid := 1, [1450].log_data[8].valid := 1, [1450].log_data[9].valid := 1, [1450].log_data[10].valid := 1, [1450].log_data[11].valid := 1, [1450].log_data[12].valid := 1, [1450].log_data[13].valid := 1, [1450].log_data[14].valid := 1, [1450].log_data[15].valid := 1, [1450].log_data[16].valid := 1, [1450].log_data[17].valid := 1, [1450].log_data[18].valid := 1, [1450].log_data[19].valid := 1, [1450].time.Year := 2023, [1450].time.Month := 1, [1450].time.Day := 14, [1450].time.Hour := 17, [1450].time.Minute := 14, [1450].time.Second := 59, [1451].log_data[0].min := 1.0, [1451].log_data[0].max := 1.0, [1451].log_data[0].total := 300.0, [1451].log_data[0].time := 300.0, [1451].log_data[0].minminute := 15, [1451].log_data[0].maxminute := 15, [1451].log_data[0].valid := 1, [1451].log_data[1].valid := 1, [1451].log_data[2].valid := 1, [1451].log_data[3].valid := 1, [1451].log_data[4].valid := 1, [1451].log_data[5].valid := 1,
        [1451].log_data[6].valid := 1, [1451].log_data[7].valid := 1, [1451].log_data[8].valid := 1, [1451].log_data[9].valid := 1, [1451].log_data[10].valid := 1, [1451].log_data[11].valid := 1, [1451].log_data[12].valid := 1, [1451].log_data[13].valid := 1, [1451].log_data[14].valid := 1, [1451].log_data[15].valid := 1, [1451].log_data[16].valid := 1, [1451].log_data[17].valid := 1, [1451].log_data[18].valid := 1, [1451].log_data[19].valid := 1, [1451].time.Year := 2023, [1451].time.Month := 1, [1451].time.Day := 14, [1451].time.Hour := 17, [1451].time.Minute := 19, [1451].time.Second := 59, [1452].log_data[0].min := 1.0, [1452].log_data[0].max := 1.0, [1452].log_data[0].total := 300.0, [1452].log_data[0].time := 300.0, [1452].log_data[0].minminute := 20, [1452].log_data[0].maxminute := 20, [1452].log_data[0].valid := 1, [1452].log_data[1].valid := 1, [1452].log_data[2].valid := 1, [1452].log_data[3].valid := 1, [1452].log_data[4].valid := 1, [1452].log_data[5].valid := 1, [1452].log_data[6].valid := 1, [1452].log_data[7].valid := 1, [1452].log_data[8].valid := 1, [1452].log_data[9].valid := 1, [1452].log_data[10].valid := 1, [1452].log_data[11].valid := 1, [1452].log_data[12].valid := 1, [1452].log_data[13].valid := 1, [1452].log_data[14].valid := 1, [1452].log_data[15].valid := 1, [1452].log_data[16].valid := 1, [1452].log_data[17].valid := 1, [1452].log_data[18].valid := 1, [1452].log_data[19].valid := 1, [1452].time.Year := 2023, [1452].time.Month := 1, [1452].time.Day := 14, [1452].time.Hour := 17, [1452].time.Minute := 24, [1452].time.Second := 59, [1453].log_data[0].min := 1.0, [1453].log_data[0].max := 1.0, [1453].log_data[0].total := 300.0, [1453].log_data[0].time := 300.0, [1453].log_data[0].minminute := 25, [1453].log_data[0].maxminute := 25, [1453].log_data[0].valid := 1, [1453].log_data[1].valid := 1,
        [1453].log_data[2].valid := 1, [1453].log_data[3].valid := 1, [1453].log_data[4].valid := 1, [1453].log_data[5].valid := 1, [1453].log_data[6].valid := 1, [1453].log_data[7].valid := 1, [1453].log_data[8].valid := 1, [1453].log_data[9].valid := 1, [1453].log_data[10].valid := 1, [1453].log_data[11].valid := 1, [1453].log_data[12].valid := 1, [1453].log_data[13].valid := 1, [1453].log_data[14].valid := 1, [1453].log_data[15].valid := 1, [1453].log_data[16].valid := 1, [1453].log_data[17].valid := 1, [1453].log_data[18].valid := 1, [1453].log_data[19].valid := 1, [1453].time.Year := 2023, [1453].time.Month := 1, [1453].time.Day := 14, [1453].time.Hour := 17, [1453].time.Minute := 29, [1453].time.Second := 59, [1454].log_data[0].min := 1.0, [1454].log_data[0].max := 1.0, [1454].log_data[0].total := 300.0, [1454].log_data[0].time := 300.0, [1454].log_data[0].minminute := 30, [1454].log_data[0].maxminute := 30, [1454].log_data[0].valid := 1, [1454].log_data[1].valid := 1, [1454].log_data[2].valid := 1, [1454].log_data[3].valid := 1, [1454].log_data[4].valid := 1, [1454].log_data[5].valid := 1, [1454].log_data[6].valid := 1, [1454].log_data[7].valid := 1, [1454].log_data[8].valid := 1, [1454].log_data[9].valid := 1, [1454].log_data[10].valid := 1, [1454].log_data[11].valid := 1, [1454].log_data[12].valid := 1, [1454].log_data[13].valid := 1, [1454].log_data[14].valid := 1, [1454].log_data[15].valid := 1, [1454].log_data[16].valid := 1, [1454].log_data[17].valid := 1, [1454].log_data[18].valid := 1, [1454].log_data[19].valid := 1, [1454].time.Year := 2023, [1454].time.Month := 1, [1454].time.Day := 14, [1454].time.Hour := 17, [1454].time.Minute := 34, [1454].time.Second := 59, [1455].log_data[0].min := 1.0, [1455].log_data[0].max := 1.0, [1455].log_data[0].total := 300.0, [1455].log_data[0].time := 300.0,
        [1455].log_data[0].minminute := 35, [1455].log_data[0].maxminute := 35, [1455].log_data[0].valid := 1, [1455].log_data[1].valid := 1, [1455].log_data[2].valid := 1, [1455].log_data[3].valid := 1, [1455].log_data[4].valid := 1, [1455].log_data[5].valid := 1, [1455].log_data[6].valid := 1, [1455].log_data[7].valid := 1, [1455].log_data[8].valid := 1, [1455].log_data[9].valid := 1, [1455].log_data[10].valid := 1, [1455].log_data[11].valid := 1, [1455].log_data[12].valid := 1, [1455].log_data[13].valid := 1, [1455].log_data[14].valid := 1, [1455].log_data[15].valid := 1, [1455].log_data[16].valid := 1, [1455].log_data[17].valid := 1, [1455].log_data[18].valid := 1, [1455].log_data[19].valid := 1, [1455].time.Year := 2023, [1455].time.Month := 1, [1455].time.Day := 14, [1455].time.Hour := 17, [1455].time.Minute := 39, [1455].time.Second := 59, [1456].log_data[0].min := 1.0, [1456].log_data[0].max := 1.0, [1456].log_data[0].total := 300.0, [1456].log_data[0].time := 300.0, [1456].log_data[0].minminute := 40, [1456].log_data[0].maxminute := 40, [1456].log_data[0].valid := 1, [1456].log_data[1].valid := 1, [1456].log_data[2].valid := 1, [1456].log_data[3].valid := 1, [1456].log_data[4].valid := 1, [1456].log_data[5].valid := 1, [1456].log_data[6].valid := 1, [1456].log_data[7].valid := 1, [1456].log_data[8].valid := 1, [1456].log_data[9].valid := 1, [1456].log_data[10].valid := 1, [1456].log_data[11].valid := 1, [1456].log_data[12].valid := 1, [1456].log_data[13].valid := 1, [1456].log_data[14].valid := 1, [1456].log_data[15].valid := 1, [1456].log_data[16].valid := 1, [1456].log_data[17].valid := 1, [1456].log_data[18].valid := 1, [1456].log_data[19].valid := 1, [1456].time.Year := 2023, [1456].time.Month := 1, [1456].time.Day := 14, [1456].time.Hour := 17, [1456].time.Minute := 44, [1456].time.Second := 59,
        [1457].log_data[0].min := 1.0, [1457].log_data[0].max := 1.0, [1457].log_data[0].total := 300.0, [1457].log_data[0].time := 300.0, [1457].log_data[0].minminute := 45, [1457].log_data[0].maxminute := 45, [1457].log_data[0].valid := 1, [1457].log_data[1].valid := 1, [1457].log_data[2].valid := 1, [1457].log_data[3].valid := 1, [1457].log_data[4].valid := 1, [1457].log_data[5].valid := 1, [1457].log_data[6].valid := 1, [1457].log_data[7].valid := 1, [1457].log_data[8].valid := 1, [1457].log_data[9].valid := 1, [1457].log_data[10].valid := 1, [1457].log_data[11].valid := 1, [1457].log_data[12].valid := 1, [1457].log_data[13].valid := 1, [1457].log_data[14].valid := 1, [1457].log_data[15].valid := 1, [1457].log_data[16].valid := 1, [1457].log_data[17].valid := 1, [1457].log_data[18].valid := 1, [1457].log_data[19].valid := 1, [1457].time.Year := 2023, [1457].time.Month := 1, [1457].time.Day := 14, [1457].time.Hour := 17, [1457].time.Minute := 49, [1457].time.Second := 59, [1458].log_data[0].min := 1.0, [1458].log_data[0].max := 1.0, [1458].log_data[0].total := 300.0, [1458].log_data[0].time := 300.0, [1458].log_data[0].minminute := 50, [1458].log_data[0].maxminute := 50, [1458].log_data[0].valid := 1, [1458].log_data[1].valid := 1, [1458].log_data[2].valid := 1, [1458].log_data[3].valid := 1, [1458].log_data[4].valid := 1, [1458].log_data[5].valid := 1, [1458].log_data[6].valid := 1, [1458].log_data[7].valid := 1, [1458].log_data[8].valid := 1, [1458].log_data[9].valid := 1, [1458].log_data[10].valid := 1, [1458].log_data[11].valid := 1, [1458].log_data[12].valid := 1, [1458].log_data[13].valid := 1, [1458].log_data[14].valid := 1, [1458].log_data[15].valid := 1, [1458].log_data[16].valid := 1, [1458].log_data[17].valid := 1, [1458].log_data[18].valid := 1, [1458].log_data[19].valid := 1, [1458].time.Year := 2023, [1458].time.Month := 1,
        [1458].time.Day := 14, [1458].time.Hour := 17, [1458].time.Minute := 54, [1458].time.Second := 59, [1459].log_data[0].min := 1.0, [1459].log_data[0].max := 1.0, [1459].log_data[0].total := 300.0, [1459].log_data[0].time := 300.0, [1459].log_data[0].minminute := 55, [1459].log_data[0].maxminute := 55, [1459].log_data[0].valid := 1, [1459].log_data[1].valid := 1, [1459].log_data[2].valid := 1, [1459].log_data[3].valid := 1, [1459].log_data[4].valid := 1, [1459].log_data[5].valid := 1, [1459].log_data[6].valid := 1, [1459].log_data[7].valid := 1, [1459].log_data[8].valid := 1, [1459].log_data[9].valid := 1, [1459].log_data[10].valid := 1, [1459].log_data[11].valid := 1, [1459].log_data[12].valid := 1, [1459].log_data[13].valid := 1, [1459].log_data[14].valid := 1, [1459].log_data[15].valid := 1, [1459].log_data[16].valid := 1, [1459].log_data[17].valid := 1, [1459].log_data[18].valid := 1, [1459].log_data[19].valid := 1, [1459].time.Year := 2023, [1459].time.Month := 1, [1459].time.Day := 14, [1459].time.Hour := 17, [1459].time.Minute := 59, [1459].time.Second := 59, [1460].log_data[0].min := 1.0, [1460].log_data[0].max := 1.0, [1460].log_data[0].total := 300.0, [1460].log_data[0].time := 300.0, [1460].log_data[0].valid := 1, [1460].log_data[1].valid := 1, [1460].log_data[2].valid := 1, [1460].log_data[3].valid := 1, [1460].log_data[4].valid := 1, [1460].log_data[5].valid := 1, [1460].log_data[6].valid := 1, [1460].log_data[7].valid := 1, [1460].log_data[8].valid := 1, [1460].log_data[9].valid := 1, [1460].log_data[10].valid := 1, [1460].log_data[11].valid := 1, [1460].log_data[12].valid := 1, [1460].log_data[13].valid := 1, [1460].log_data[14].valid := 1, [1460].log_data[15].valid := 1, [1460].log_data[16].valid := 1, [1460].log_data[17].valid := 1, [1460].log_data[18].valid := 1, [1460].log_data[19].valid := 1,
        [1460].time.Year := 2023, [1460].time.Month := 1, [1460].time.Day := 14, [1460].time.Hour := 18, [1460].time.Minute := 4, [1460].time.Second := 59, [1461].log_data[0].min := 1.0, [1461].log_data[0].max := 1.0, [1461].log_data[0].total := 300.0, [1461].log_data[0].time := 300.0, [1461].log_data[0].minminute := 5, [1461].log_data[0].maxminute := 5, [1461].log_data[0].valid := 1, [1461].log_data[1].valid := 1, [1461].log_data[2].valid := 1, [1461].log_data[3].valid := 1, [1461].log_data[4].valid := 1, [1461].log_data[5].valid := 1, [1461].log_data[6].valid := 1, [1461].log_data[7].valid := 1, [1461].log_data[8].valid := 1, [1461].log_data[9].valid := 1, [1461].log_data[10].valid := 1, [1461].log_data[11].valid := 1, [1461].log_data[12].valid := 1, [1461].log_data[13].valid := 1, [1461].log_data[14].valid := 1, [1461].log_data[15].valid := 1, [1461].log_data[16].valid := 1, [1461].log_data[17].valid := 1, [1461].log_data[18].valid := 1, [1461].log_data[19].valid := 1, [1461].time.Year := 2023, [1461].time.Month := 1, [1461].time.Day := 14, [1461].time.Hour := 18, [1461].time.Minute := 9, [1461].time.Second := 59, [1462].log_data[0].min := 1.0, [1462].log_data[0].max := 1.0, [1462].log_data[0].total := 300.0, [1462].log_data[0].time := 300.0, [1462].log_data[0].minminute := 10, [1462].log_data[0].maxminute := 10, [1462].log_data[0].valid := 1, [1462].log_data[1].valid := 1, [1462].log_data[2].valid := 1, [1462].log_data[3].valid := 1, [1462].log_data[4].valid := 1, [1462].log_data[5].valid := 1, [1462].log_data[6].valid := 1, [1462].log_data[7].valid := 1, [1462].log_data[8].valid := 1, [1462].log_data[9].valid := 1, [1462].log_data[10].valid := 1, [1462].log_data[11].valid := 1, [1462].log_data[12].valid := 1, [1462].log_data[13].valid := 1, [1462].log_data[14].valid := 1, [1462].log_data[15].valid := 1,
        [1462].log_data[16].valid := 1, [1462].log_data[17].valid := 1, [1462].log_data[18].valid := 1, [1462].log_data[19].valid := 1, [1462].time.Year := 2023, [1462].time.Month := 1, [1462].time.Day := 14, [1462].time.Hour := 18, [1462].time.Minute := 14, [1462].time.Second := 59, [1463].log_data[0].min := 1.0, [1463].log_data[0].max := 1.0, [1463].log_data[0].total := 300.0, [1463].log_data[0].time := 300.0, [1463].log_data[0].minminute := 15, [1463].log_data[0].maxminute := 15, [1463].log_data[0].valid := 1, [1463].log_data[1].valid := 1, [1463].log_data[2].valid := 1, [1463].log_data[3].valid := 1, [1463].log_data[4].valid := 1, [1463].log_data[5].valid := 1, [1463].log_data[6].valid := 1, [1463].log_data[7].valid := 1, [1463].log_data[8].valid := 1, [1463].log_data[9].valid := 1, [1463].log_data[10].valid := 1, [1463].log_data[11].valid := 1, [1463].log_data[12].valid := 1, [1463].log_data[13].valid := 1, [1463].log_data[14].valid := 1, [1463].log_data[15].valid := 1, [1463].log_data[16].valid := 1, [1463].log_data[17].valid := 1, [1463].log_data[18].valid := 1, [1463].log_data[19].valid := 1, [1463].time.Year := 2023, [1463].time.Month := 1, [1463].time.Day := 14, [1463].time.Hour := 18, [1463].time.Minute := 19, [1463].time.Second := 59, [1464].log_data[0].min := 1.0, [1464].log_data[0].max := 1.0, [1464].log_data[0].total := 300.0, [1464].log_data[0].time := 300.0, [1464].log_data[0].minminute := 20, [1464].log_data[0].maxminute := 20, [1464].log_data[0].valid := 1, [1464].log_data[1].valid := 1, [1464].log_data[2].valid := 1, [1464].log_data[3].valid := 1, [1464].log_data[4].valid := 1, [1464].log_data[5].valid := 1, [1464].log_data[6].valid := 1, [1464].log_data[7].valid := 1, [1464].log_data[8].valid := 1, [1464].log_data[9].valid := 1, [1464].log_data[10].valid := 1, [1464].log_data[11].valid := 1,
        [1464].log_data[12].valid := 1, [1464].log_data[13].valid := 1, [1464].log_data[14].valid := 1, [1464].log_data[15].valid := 1, [1464].log_data[16].valid := 1, [1464].log_data[17].valid := 1, [1464].log_data[18].valid := 1, [1464].log_data[19].valid := 1, [1464].time.Year := 2023, [1464].time.Month := 1, [1464].time.Day := 14, [1464].time.Hour := 18, [1464].time.Minute := 24, [1464].time.Second := 59, [1465].log_data[0].min := 1.0, [1465].log_data[0].max := 1.0, [1465].log_data[0].total := 300.0, [1465].log_data[0].time := 300.0, [1465].log_data[0].minminute := 25, [1465].log_data[0].maxminute := 25, [1465].log_data[0].valid := 1, [1465].log_data[1].valid := 1, [1465].log_data[2].valid := 1, [1465].log_data[3].valid := 1, [1465].log_data[4].valid := 1, [1465].log_data[5].valid := 1, [1465].log_data[6].valid := 1, [1465].log_data[7].valid := 1, [1465].log_data[8].valid := 1, [1465].log_data[9].valid := 1, [1465].log_data[10].valid := 1, [1465].log_data[11].valid := 1, [1465].log_data[12].valid := 1, [1465].log_data[13].valid := 1, [1465].log_data[14].valid := 1, [1465].log_data[15].valid := 1, [1465].log_data[16].valid := 1, [1465].log_data[17].valid := 1, [1465].log_data[18].valid := 1, [1465].log_data[19].valid := 1, [1465].time.Year := 2023, [1465].time.Month := 1, [1465].time.Day := 14, [1465].time.Hour := 18, [1465].time.Minute := 29, [1465].time.Second := 59, [1466].log_data[0].min := 1.0, [1466].log_data[0].max := 1.0, [1466].log_data[0].total := 300.0, [1466].log_data[0].time := 300.0, [1466].log_data[0].minminute := 30, [1466].log_data[0].maxminute := 30, [1466].log_data[0].valid := 1, [1466].log_data[1].valid := 1, [1466].log_data[2].valid := 1, [1466].log_data[3].valid := 1, [1466].log_data[4].valid := 1, [1466].log_data[5].valid := 1, [1466].log_data[6].valid := 1, [1466].log_data[7].valid := 1,
        [1466].log_data[8].valid := 1, [1466].log_data[9].valid := 1, [1466].log_data[10].valid := 1, [1466].log_data[11].valid := 1, [1466].log_data[12].valid := 1, [1466].log_data[13].valid := 1, [1466].log_data[14].valid := 1, [1466].log_data[15].valid := 1, [1466].log_data[16].valid := 1, [1466].log_data[17].valid := 1, [1466].log_data[18].valid := 1, [1466].log_data[19].valid := 1, [1466].time.Year := 2023, [1466].time.Month := 1, [1466].time.Day := 14, [1466].time.Hour := 18, [1466].time.Minute := 34, [1466].time.Second := 59, [1467].log_data[0].min := 1.0, [1467].log_data[0].max := 1.0, [1467].log_data[0].total := 300.0, [1467].log_data[0].time := 300.0, [1467].log_data[0].minminute := 35, [1467].log_data[0].maxminute := 35, [1467].log_data[0].valid := 1, [1467].log_data[1].valid := 1, [1467].log_data[2].valid := 1, [1467].log_data[3].valid := 1, [1467].log_data[4].valid := 1, [1467].log_data[5].valid := 1, [1467].log_data[6].valid := 1, [1467].log_data[7].valid := 1, [1467].log_data[8].valid := 1, [1467].log_data[9].valid := 1, [1467].log_data[10].valid := 1, [1467].log_data[11].valid := 1, [1467].log_data[12].valid := 1, [1467].log_data[13].valid := 1, [1467].log_data[14].valid := 1, [1467].log_data[15].valid := 1, [1467].log_data[16].valid := 1, [1467].log_data[17].valid := 1, [1467].log_data[18].valid := 1, [1467].log_data[19].valid := 1, [1467].time.Year := 2023, [1467].time.Month := 1, [1467].time.Day := 14, [1467].time.Hour := 18, [1467].time.Minute := 39, [1467].time.Second := 59, [1468].log_data[0].min := 1.0, [1468].log_data[0].max := 1.0, [1468].log_data[0].total := 300.0, [1468].log_data[0].time := 300.0, [1468].log_data[0].minminute := 40, [1468].log_data[0].maxminute := 40, [1468].log_data[0].valid := 1, [1468].log_data[1].valid := 1, [1468].log_data[2].valid := 1, [1468].log_data[3].valid := 1,
        [1468].log_data[4].valid := 1, [1468].log_data[5].valid := 1, [1468].log_data[6].valid := 1, [1468].log_data[7].valid := 1, [1468].log_data[8].valid := 1, [1468].log_data[9].valid := 1, [1468].log_data[10].valid := 1, [1468].log_data[11].valid := 1, [1468].log_data[12].valid := 1, [1468].log_data[13].valid := 1, [1468].log_data[14].valid := 1, [1468].log_data[15].valid := 1, [1468].log_data[16].valid := 1, [1468].log_data[17].valid := 1, [1468].log_data[18].valid := 1, [1468].log_data[19].valid := 1, [1468].time.Year := 2023, [1468].time.Month := 1, [1468].time.Day := 14, [1468].time.Hour := 18, [1468].time.Minute := 44, [1468].time.Second := 59, [1469].log_data[0].min := 1.0, [1469].log_data[0].max := 1.0, [1469].log_data[0].total := 300.0, [1469].log_data[0].time := 300.0, [1469].log_data[0].minminute := 45, [1469].log_data[0].maxminute := 45, [1469].log_data[0].valid := 1, [1469].log_data[1].valid := 1, [1469].log_data[2].valid := 1, [1469].log_data[3].valid := 1, [1469].log_data[4].valid := 1, [1469].log_data[5].valid := 1, [1469].log_data[6].valid := 1, [1469].log_data[7].valid := 1, [1469].log_data[8].valid := 1, [1469].log_data[9].valid := 1, [1469].log_data[10].valid := 1, [1469].log_data[11].valid := 1, [1469].log_data[12].valid := 1, [1469].log_data[13].valid := 1, [1469].log_data[14].valid := 1, [1469].log_data[15].valid := 1, [1469].log_data[16].valid := 1, [1469].log_data[17].valid := 1, [1469].log_data[18].valid := 1, [1469].log_data[19].valid := 1, [1469].time.Year := 2023, [1469].time.Month := 1, [1469].time.Day := 14, [1469].time.Hour := 18, [1469].time.Minute := 49, [1469].time.Second := 59, [1470].log_data[0].min := 1.0, [1470].log_data[0].max := 1.0, [1470].log_data[0].total := 300.0, [1470].log_data[0].time := 300.0, [1470].log_data[0].minminute := 50, [1470].log_data[0].maxminute := 50,
        [1470].log_data[0].valid := 1, [1470].log_data[1].valid := 1, [1470].log_data[2].valid := 1, [1470].log_data[3].valid := 1, [1470].log_data[4].valid := 1, [1470].log_data[5].valid := 1, [1470].log_data[6].valid := 1, [1470].log_data[7].valid := 1, [1470].log_data[8].valid := 1, [1470].log_data[9].valid := 1, [1470].log_data[10].valid := 1, [1470].log_data[11].valid := 1, [1470].log_data[12].valid := 1, [1470].log_data[13].valid := 1, [1470].log_data[14].valid := 1, [1470].log_data[15].valid := 1, [1470].log_data[16].valid := 1, [1470].log_data[17].valid := 1, [1470].log_data[18].valid := 1, [1470].log_data[19].valid := 1, [1470].time.Year := 2023, [1470].time.Month := 1, [1470].time.Day := 14, [1470].time.Hour := 18, [1470].time.Minute := 54, [1470].time.Second := 59, [1471].log_data[0].min := 1.0, [1471].log_data[0].max := 1.0, [1471].log_data[0].total := 300.0, [1471].log_data[0].time := 300.0, [1471].log_data[0].minminute := 55, [1471].log_data[0].maxminute := 55, [1471].log_data[0].valid := 1, [1471].log_data[1].valid := 1, [1471].log_data[2].valid := 1, [1471].log_data[3].valid := 1, [1471].log_data[4].valid := 1, [1471].log_data[5].valid := 1, [1471].log_data[6].valid := 1, [1471].log_data[7].valid := 1, [1471].log_data[8].valid := 1, [1471].log_data[9].valid := 1, [1471].log_data[10].valid := 1, [1471].log_data[11].valid := 1, [1471].log_data[12].valid := 1, [1471].log_data[13].valid := 1, [1471].log_data[14].valid := 1, [1471].log_data[15].valid := 1, [1471].log_data[16].valid := 1, [1471].log_data[17].valid := 1, [1471].log_data[18].valid := 1, [1471].log_data[19].valid := 1, [1471].time.Year := 2023, [1471].time.Month := 1, [1471].time.Day := 14, [1471].time.Hour := 18, [1471].time.Minute := 59, [1471].time.Second := 59, [1472].log_data[0].min := 1.0, [1472].log_data[0].max := 1.0,
        [1472].log_data[0].total := 300.0, [1472].log_data[0].time := 300.0, [1472].log_data[0].valid := 1, [1472].log_data[1].valid := 1, [1472].log_data[2].valid := 1, [1472].log_data[3].valid := 1, [1472].log_data[4].valid := 1, [1472].log_data[5].valid := 1, [1472].log_data[6].valid := 1, [1472].log_data[7].valid := 1, [1472].log_data[8].valid := 1, [1472].log_data[9].valid := 1, [1472].log_data[10].valid := 1, [1472].log_data[11].valid := 1, [1472].log_data[12].valid := 1, [1472].log_data[13].valid := 1, [1472].log_data[14].valid := 1, [1472].log_data[15].valid := 1, [1472].log_data[16].valid := 1, [1472].log_data[17].valid := 1, [1472].log_data[18].valid := 1, [1472].log_data[19].valid := 1, [1472].time.Year := 2023, [1472].time.Month := 1, [1472].time.Day := 14, [1472].time.Hour := 19, [1472].time.Minute := 4, [1472].time.Second := 59, [1473].log_data[0].min := 1.0, [1473].log_data[0].max := 1.0, [1473].log_data[0].total := 300.0, [1473].log_data[0].time := 300.0, [1473].log_data[0].minminute := 5, [1473].log_data[0].maxminute := 5, [1473].log_data[0].valid := 1, [1473].log_data[1].valid := 1, [1473].log_data[2].valid := 1, [1473].log_data[3].valid := 1, [1473].log_data[4].valid := 1, [1473].log_data[5].valid := 1, [1473].log_data[6].valid := 1, [1473].log_data[7].valid := 1, [1473].log_data[8].valid := 1, [1473].log_data[9].valid := 1, [1473].log_data[10].valid := 1, [1473].log_data[11].valid := 1, [1473].log_data[12].valid := 1, [1473].log_data[13].valid := 1, [1473].log_data[14].valid := 1, [1473].log_data[15].valid := 1, [1473].log_data[16].valid := 1, [1473].log_data[17].valid := 1, [1473].log_data[18].valid := 1, [1473].log_data[19].valid := 1, [1473].time.Year := 2023, [1473].time.Month := 1, [1473].time.Day := 14, [1473].time.Hour := 19, [1473].time.Minute := 9, [1473].time.Second := 59,
        [1474].log_data[0].min := 1.0, [1474].log_data[0].max := 1.0, [1474].log_data[0].total := 300.0, [1474].log_data[0].time := 300.0, [1474].log_data[0].minminute := 10, [1474].log_data[0].maxminute := 10, [1474].log_data[0].valid := 1, [1474].log_data[1].valid := 1, [1474].log_data[2].valid := 1, [1474].log_data[3].valid := 1, [1474].log_data[4].valid := 1, [1474].log_data[5].valid := 1, [1474].log_data[6].valid := 1, [1474].log_data[7].valid := 1, [1474].log_data[8].valid := 1, [1474].log_data[9].valid := 1, [1474].log_data[10].valid := 1, [1474].log_data[11].valid := 1, [1474].log_data[12].valid := 1, [1474].log_data[13].valid := 1, [1474].log_data[14].valid := 1, [1474].log_data[15].valid := 1, [1474].log_data[16].valid := 1, [1474].log_data[17].valid := 1, [1474].log_data[18].valid := 1, [1474].log_data[19].valid := 1, [1474].time.Year := 2023, [1474].time.Month := 1, [1474].time.Day := 14, [1474].time.Hour := 19, [1474].time.Minute := 14, [1474].time.Second := 59, [1475].log_data[0].min := 1.0, [1475].log_data[0].max := 1.0, [1475].log_data[0].total := 300.0, [1475].log_data[0].time := 300.0, [1475].log_data[0].minminute := 15, [1475].log_data[0].maxminute := 15, [1475].log_data[0].valid := 1, [1475].log_data[1].valid := 1, [1475].log_data[2].valid := 1, [1475].log_data[3].valid := 1, [1475].log_data[4].valid := 1, [1475].log_data[5].valid := 1, [1475].log_data[6].valid := 1, [1475].log_data[7].valid := 1, [1475].log_data[8].valid := 1, [1475].log_data[9].valid := 1, [1475].log_data[10].valid := 1, [1475].log_data[11].valid := 1, [1475].log_data[12].valid := 1, [1475].log_data[13].valid := 1, [1475].log_data[14].valid := 1, [1475].log_data[15].valid := 1, [1475].log_data[16].valid := 1, [1475].log_data[17].valid := 1, [1475].log_data[18].valid := 1, [1475].log_data[19].valid := 1, [1475].time.Year := 2023, [1475].time.Month := 1,
        [1475].time.Day := 14, [1475].time.Hour := 19, [1475].time.Minute := 19, [1475].time.Second := 59, [1476].log_data[0].min := 1.0, [1476].log_data[0].max := 1.0, [1476].log_data[0].total := 300.0, [1476].log_data[0].time := 300.0, [1476].log_data[0].minminute := 20, [1476].log_data[0].maxminute := 20, [1476].log_data[0].valid := 1, [1476].log_data[1].valid := 1, [1476].log_data[2].valid := 1, [1476].log_data[3].valid := 1, [1476].log_data[4].valid := 1, [1476].log_data[5].valid := 1, [1476].log_data[6].valid := 1, [1476].log_data[7].valid := 1, [1476].log_data[8].valid := 1, [1476].log_data[9].valid := 1, [1476].log_data[10].valid := 1, [1476].log_data[11].valid := 1, [1476].log_data[12].valid := 1, [1476].log_data[13].valid := 1, [1476].log_data[14].valid := 1, [1476].log_data[15].valid := 1, [1476].log_data[16].valid := 1, [1476].log_data[17].valid := 1, [1476].log_data[18].valid := 1, [1476].log_data[19].valid := 1, [1476].time.Year := 2023, [1476].time.Month := 1, [1476].time.Day := 14, [1476].time.Hour := 19, [1476].time.Minute := 24, [1476].time.Second := 59, [1477].log_data[0].min := 1.0, [1477].log_data[0].max := 1.0, [1477].log_data[0].total := 300.0, [1477].log_data[0].time := 300.0, [1477].log_data[0].minminute := 25, [1477].log_data[0].maxminute := 25, [1477].log_data[0].valid := 1, [1477].log_data[1].valid := 1, [1477].log_data[2].valid := 1, [1477].log_data[3].valid := 1, [1477].log_data[4].valid := 1, [1477].log_data[5].valid := 1, [1477].log_data[6].valid := 1, [1477].log_data[7].valid := 1, [1477].log_data[8].valid := 1, [1477].log_data[9].valid := 1, [1477].log_data[10].valid := 1, [1477].log_data[11].valid := 1, [1477].log_data[12].valid := 1, [1477].log_data[13].valid := 1, [1477].log_data[14].valid := 1, [1477].log_data[15].valid := 1, [1477].log_data[16].valid := 1, [1477].log_data[17].valid := 1,
        [1477].log_data[18].valid := 1, [1477].log_data[19].valid := 1, [1477].time.Year := 2023, [1477].time.Month := 1, [1477].time.Day := 14, [1477].time.Hour := 19, [1477].time.Minute := 29, [1477].time.Second := 59, [1478].log_data[0].min := 1.0, [1478].log_data[0].max := 1.0, [1478].log_data[0].total := 300.0, [1478].log_data[0].time := 300.0, [1478].log_data[0].minminute := 30, [1478].log_data[0].maxminute := 30, [1478].log_data[0].valid := 1, [1478].log_data[1].valid := 1, [1478].log_data[2].valid := 1, [1478].log_data[3].valid := 1, [1478].log_data[4].valid := 1, [1478].log_data[5].valid := 1, [1478].log_data[6].valid := 1, [1478].log_data[7].valid := 1, [1478].log_data[8].valid := 1, [1478].log_data[9].valid := 1, [1478].log_data[10].valid := 1, [1478].log_data[11].valid := 1, [1478].log_data[12].valid := 1, [1478].log_data[13].valid := 1, [1478].log_data[14].valid := 1, [1478].log_data[15].valid := 1, [1478].log_data[16].valid := 1, [1478].log_data[17].valid := 1, [1478].log_data[18].valid := 1, [1478].log_data[19].valid := 1, [1478].time.Year := 2023, [1478].time.Month := 1, [1478].time.Day := 14, [1478].time.Hour := 19, [1478].time.Minute := 34, [1478].time.Second := 59, [1479].log_data[0].min := 1.0, [1479].log_data[0].max := 1.0, [1479].log_data[0].total := 300.0, [1479].log_data[0].time := 300.0, [1479].log_data[0].minminute := 35, [1479].log_data[0].maxminute := 35, [1479].log_data[0].valid := 1, [1479].log_data[1].valid := 1, [1479].log_data[2].valid := 1, [1479].log_data[3].valid := 1, [1479].log_data[4].valid := 1, [1479].log_data[5].valid := 1, [1479].log_data[6].valid := 1, [1479].log_data[7].valid := 1, [1479].log_data[8].valid := 1, [1479].log_data[9].valid := 1, [1479].log_data[10].valid := 1, [1479].log_data[11].valid := 1, [1479].log_data[12].valid := 1, [1479].log_data[13].valid := 1,
        [1479].log_data[14].valid := 1, [1479].log_data[15].valid := 1, [1479].log_data[16].valid := 1, [1479].log_data[17].valid := 1, [1479].log_data[18].valid := 1, [1479].log_data[19].valid := 1, [1479].time.Year := 2023, [1479].time.Month := 1, [1479].time.Day := 14, [1479].time.Hour := 19, [1479].time.Minute := 39, [1479].time.Second := 59, [1480].log_data[0].min := 1.0, [1480].log_data[0].max := 1.0, [1480].log_data[0].total := 300.0, [1480].log_data[0].time := 300.0, [1480].log_data[0].minminute := 40, [1480].log_data[0].maxminute := 40, [1480].log_data[0].valid := 1, [1480].log_data[1].valid := 1, [1480].log_data[2].valid := 1, [1480].log_data[3].valid := 1, [1480].log_data[4].valid := 1, [1480].log_data[5].valid := 1, [1480].log_data[6].valid := 1, [1480].log_data[7].valid := 1, [1480].log_data[8].valid := 1, [1480].log_data[9].valid := 1, [1480].log_data[10].valid := 1, [1480].log_data[11].valid := 1, [1480].log_data[12].valid := 1, [1480].log_data[13].valid := 1, [1480].log_data[14].valid := 1, [1480].log_data[15].valid := 1, [1480].log_data[16].valid := 1, [1480].log_data[17].valid := 1, [1480].log_data[18].valid := 1, [1480].log_data[19].valid := 1, [1480].time.Year := 2023, [1480].time.Month := 1, [1480].time.Day := 14, [1480].time.Hour := 19, [1480].time.Minute := 44, [1480].time.Second := 59, [1481].log_data[0].min := 1.0, [1481].log_data[0].max := 1.0, [1481].log_data[0].total := 300.0, [1481].log_data[0].time := 300.0, [1481].log_data[0].minminute := 45, [1481].log_data[0].maxminute := 45, [1481].log_data[0].valid := 1, [1481].log_data[1].valid := 1, [1481].log_data[2].valid := 1, [1481].log_data[3].valid := 1, [1481].log_data[4].valid := 1, [1481].log_data[5].valid := 1, [1481].log_data[6].valid := 1, [1481].log_data[7].valid := 1, [1481].log_data[8].valid := 1, [1481].log_data[9].valid := 1,
        [1481].log_data[10].valid := 1, [1481].log_data[11].valid := 1, [1481].log_data[12].valid := 1, [1481].log_data[13].valid := 1, [1481].log_data[14].valid := 1, [1481].log_data[15].valid := 1, [1481].log_data[16].valid := 1, [1481].log_data[17].valid := 1, [1481].log_data[18].valid := 1, [1481].log_data[19].valid := 1, [1481].time.Year := 2023, [1481].time.Month := 1, [1481].time.Day := 14, [1481].time.Hour := 19, [1481].time.Minute := 49, [1481].time.Second := 59, [1482].log_data[0].min := 1.0, [1482].log_data[0].max := 1.0, [1482].log_data[0].total := 300.0, [1482].log_data[0].time := 300.0, [1482].log_data[0].minminute := 50, [1482].log_data[0].maxminute := 50, [1482].log_data[0].valid := 1, [1482].log_data[1].valid := 1, [1482].log_data[2].valid := 1, [1482].log_data[3].valid := 1, [1482].log_data[4].valid := 1, [1482].log_data[5].valid := 1, [1482].log_data[6].valid := 1, [1482].log_data[7].valid := 1, [1482].log_data[8].valid := 1, [1482].log_data[9].valid := 1, [1482].log_data[10].valid := 1, [1482].log_data[11].valid := 1, [1482].log_data[12].valid := 1, [1482].log_data[13].valid := 1, [1482].log_data[14].valid := 1, [1482].log_data[15].valid := 1, [1482].log_data[16].valid := 1, [1482].log_data[17].valid := 1, [1482].log_data[18].valid := 1, [1482].log_data[19].valid := 1, [1482].time.Year := 2023, [1482].time.Month := 1, [1482].time.Day := 14, [1482].time.Hour := 19, [1482].time.Minute := 54, [1482].time.Second := 59, [1483].log_data[0].min := 1.0, [1483].log_data[0].max := 1.0, [1483].log_data[0].total := 300.0, [1483].log_data[0].time := 300.0, [1483].log_data[0].minminute := 55, [1483].log_data[0].maxminute := 55, [1483].log_data[0].valid := 1, [1483].log_data[1].valid := 1, [1483].log_data[2].valid := 1, [1483].log_data[3].valid := 1, [1483].log_data[4].valid := 1, [1483].log_data[5].valid := 1,
        [1483].log_data[6].valid := 1, [1483].log_data[7].valid := 1, [1483].log_data[8].valid := 1, [1483].log_data[9].valid := 1, [1483].log_data[10].valid := 1, [1483].log_data[11].valid := 1, [1483].log_data[12].valid := 1, [1483].log_data[13].valid := 1, [1483].log_data[14].valid := 1, [1483].log_data[15].valid := 1, [1483].log_data[16].valid := 1, [1483].log_data[17].valid := 1, [1483].log_data[18].valid := 1, [1483].log_data[19].valid := 1, [1483].time.Year := 2023, [1483].time.Month := 1, [1483].time.Day := 14, [1483].time.Hour := 19, [1483].time.Minute := 59, [1483].time.Second := 59, [1484].log_data[0].min := 1.0, [1484].log_data[0].max := 1.0, [1484].log_data[0].total := 300.0, [1484].log_data[0].time := 300.0, [1484].log_data[0].valid := 1, [1484].log_data[1].valid := 1, [1484].log_data[2].valid := 1, [1484].log_data[3].valid := 1, [1484].log_data[4].valid := 1, [1484].log_data[5].valid := 1, [1484].log_data[6].valid := 1, [1484].log_data[7].valid := 1, [1484].log_data[8].valid := 1, [1484].log_data[9].valid := 1, [1484].log_data[10].valid := 1, [1484].log_data[11].valid := 1, [1484].log_data[12].valid := 1, [1484].log_data[13].valid := 1, [1484].log_data[14].valid := 1, [1484].log_data[15].valid := 1, [1484].log_data[16].valid := 1, [1484].log_data[17].valid := 1, [1484].log_data[18].valid := 1, [1484].log_data[19].valid := 1, [1484].time.Year := 2023, [1484].time.Month := 1, [1484].time.Day := 14, [1484].time.Hour := 20, [1484].time.Minute := 4, [1484].time.Second := 59, [1485].log_data[0].min := 1.0, [1485].log_data[0].max := 1.0, [1485].log_data[0].total := 300.0, [1485].log_data[0].time := 300.0, [1485].log_data[0].minminute := 5, [1485].log_data[0].maxminute := 5, [1485].log_data[0].valid := 1, [1485].log_data[1].valid := 1, [1485].log_data[2].valid := 1, [1485].log_data[3].valid := 1,
        [1485].log_data[4].valid := 1, [1485].log_data[5].valid := 1, [1485].log_data[6].valid := 1, [1485].log_data[7].valid := 1, [1485].log_data[8].valid := 1, [1485].log_data[9].valid := 1, [1485].log_data[10].valid := 1, [1485].log_data[11].valid := 1, [1485].log_data[12].valid := 1, [1485].log_data[13].valid := 1, [1485].log_data[14].valid := 1, [1485].log_data[15].valid := 1, [1485].log_data[16].valid := 1, [1485].log_data[17].valid := 1, [1485].log_data[18].valid := 1, [1485].log_data[19].valid := 1, [1485].time.Year := 2023, [1485].time.Month := 1, [1485].time.Day := 14, [1485].time.Hour := 20, [1485].time.Minute := 9, [1485].time.Second := 59, [1486].log_data[0].min := 1.0, [1486].log_data[0].max := 1.0, [1486].log_data[0].total := 300.0, [1486].log_data[0].time := 300.0, [1486].log_data[0].minminute := 10, [1486].log_data[0].maxminute := 10, [1486].log_data[0].valid := 1, [1486].log_data[1].valid := 1, [1486].log_data[2].valid := 1, [1486].log_data[3].valid := 1, [1486].log_data[4].valid := 1, [1486].log_data[5].valid := 1, [1486].log_data[6].valid := 1, [1486].log_data[7].valid := 1, [1486].log_data[8].valid := 1, [1486].log_data[9].valid := 1, [1486].log_data[10].valid := 1, [1486].log_data[11].valid := 1, [1486].log_data[12].valid := 1, [1486].log_data[13].valid := 1, [1486].log_data[14].valid := 1, [1486].log_data[15].valid := 1, [1486].log_data[16].valid := 1, [1486].log_data[17].valid := 1, [1486].log_data[18].valid := 1, [1486].log_data[19].valid := 1, [1486].time.Year := 2023, [1486].time.Month := 1, [1486].time.Day := 14, [1486].time.Hour := 20, [1486].time.Minute := 14, [1486].time.Second := 59, [1487].log_data[0].min := 1.0, [1487].log_data[0].max := 1.0, [1487].log_data[0].total := 300.0, [1487].log_data[0].time := 300.0, [1487].log_data[0].minminute := 15, [1487].log_data[0].maxminute := 15,
        [1487].log_data[0].valid := 1, [1487].log_data[1].valid := 1, [1487].log_data[2].valid := 1, [1487].log_data[3].valid := 1, [1487].log_data[4].valid := 1, [1487].log_data[5].valid := 1, [1487].log_data[6].valid := 1, [1487].log_data[7].valid := 1, [1487].log_data[8].valid := 1, [1487].log_data[9].valid := 1, [1487].log_data[10].valid := 1, [1487].log_data[11].valid := 1, [1487].log_data[12].valid := 1, [1487].log_data[13].valid := 1, [1487].log_data[14].valid := 1, [1487].log_data[15].valid := 1, [1487].log_data[16].valid := 1, [1487].log_data[17].valid := 1, [1487].log_data[18].valid := 1, [1487].log_data[19].valid := 1, [1487].time.Year := 2023, [1487].time.Month := 1, [1487].time.Day := 14, [1487].time.Hour := 20, [1487].time.Minute := 19, [1487].time.Second := 59, [1488].log_data[0].min := 1.0, [1488].log_data[0].max := 1.0, [1488].log_data[0].total := 300.0, [1488].log_data[0].time := 300.0, [1488].log_data[0].minminute := 20, [1488].log_data[0].maxminute := 20, [1488].log_data[0].valid := 1, [1488].log_data[1].valid := 1, [1488].log_data[2].valid := 1, [1488].log_data[3].valid := 1, [1488].log_data[4].valid := 1, [1488].log_data[5].valid := 1, [1488].log_data[6].valid := 1, [1488].log_data[7].valid := 1, [1488].log_data[8].valid := 1, [1488].log_data[9].valid := 1, [1488].log_data[10].valid := 1, [1488].log_data[11].valid := 1, [1488].log_data[12].valid := 1, [1488].log_data[13].valid := 1, [1488].log_data[14].valid := 1, [1488].log_data[15].valid := 1, [1488].log_data[16].valid := 1, [1488].log_data[17].valid := 1, [1488].log_data[18].valid := 1, [1488].log_data[19].valid := 1, [1488].time.Year := 2023, [1488].time.Month := 1, [1488].time.Day := 14, [1488].time.Hour := 20, [1488].time.Minute := 24, [1488].time.Second := 59, [1489].log_data[0].min := 1.0, [1489].log_data[0].max := 1.0,
        [1489].log_data[0].total := 300.0, [1489].log_data[0].time := 300.0, [1489].log_data[0].minminute := 25, [1489].log_data[0].maxminute := 25, [1489].log_data[0].valid := 1, [1489].log_data[1].valid := 1, [1489].log_data[2].valid := 1, [1489].log_data[3].valid := 1, [1489].log_data[4].valid := 1, [1489].log_data[5].valid := 1, [1489].log_data[6].valid := 1, [1489].log_data[7].valid := 1, [1489].log_data[8].valid := 1, [1489].log_data[9].valid := 1, [1489].log_data[10].valid := 1, [1489].log_data[11].valid := 1, [1489].log_data[12].valid := 1, [1489].log_data[13].valid := 1, [1489].log_data[14].valid := 1, [1489].log_data[15].valid := 1, [1489].log_data[16].valid := 1, [1489].log_data[17].valid := 1, [1489].log_data[18].valid := 1, [1489].log_data[19].valid := 1, [1489].time.Year := 2023, [1489].time.Month := 1, [1489].time.Day := 14, [1489].time.Hour := 20, [1489].time.Minute := 29, [1489].time.Second := 59, [1490].log_data[0].min := 1.0, [1490].log_data[0].max := 1.0, [1490].log_data[0].total := 300.0, [1490].log_data[0].time := 300.0, [1490].log_data[0].minminute := 30, [1490].log_data[0].maxminute := 30, [1490].log_data[0].valid := 1, [1490].log_data[1].valid := 1, [1490].log_data[2].valid := 1, [1490].log_data[3].valid := 1, [1490].log_data[4].valid := 1, [1490].log_data[5].valid := 1, [1490].log_data[6].valid := 1, [1490].log_data[7].valid := 1, [1490].log_data[8].valid := 1, [1490].log_data[9].valid := 1, [1490].log_data[10].valid := 1, [1490].log_data[11].valid := 1, [1490].log_data[12].valid := 1, [1490].log_data[13].valid := 1, [1490].log_data[14].valid := 1, [1490].log_data[15].valid := 1, [1490].log_data[16].valid := 1, [1490].log_data[17].valid := 1, [1490].log_data[18].valid := 1, [1490].log_data[19].valid := 1, [1490].time.Year := 2023, [1490].time.Month := 1, [1490].time.Day := 14, [1490].time.Hour := 20,
        [1490].time.Minute := 34, [1490].time.Second := 59, [1491].log_data[0].min := 1.0, [1491].log_data[0].max := 1.0, [1491].log_data[0].total := 300.0, [1491].log_data[0].time := 300.0, [1491].log_data[0].minminute := 35, [1491].log_data[0].maxminute := 35, [1491].log_data[0].valid := 1, [1491].log_data[1].valid := 1, [1491].log_data[2].valid := 1, [1491].log_data[3].valid := 1, [1491].log_data[4].valid := 1, [1491].log_data[5].valid := 1, [1491].log_data[6].valid := 1, [1491].log_data[7].valid := 1, [1491].log_data[8].valid := 1, [1491].log_data[9].valid := 1, [1491].log_data[10].valid := 1, [1491].log_data[11].valid := 1, [1491].log_data[12].valid := 1, [1491].log_data[13].valid := 1, [1491].log_data[14].valid := 1, [1491].log_data[15].valid := 1, [1491].log_data[16].valid := 1, [1491].log_data[17].valid := 1, [1491].log_data[18].valid := 1, [1491].log_data[19].valid := 1, [1491].time.Year := 2023, [1491].time.Month := 1, [1491].time.Day := 14, [1491].time.Hour := 20, [1491].time.Minute := 39, [1491].time.Second := 59, [1492].log_data[0].min := 1.0, [1492].log_data[0].max := 1.0, [1492].log_data[0].total := 300.0, [1492].log_data[0].time := 300.0, [1492].log_data[0].minminute := 40, [1492].log_data[0].maxminute := 40, [1492].log_data[0].valid := 1, [1492].log_data[1].valid := 1, [1492].log_data[2].valid := 1, [1492].log_data[3].valid := 1, [1492].log_data[4].valid := 1, [1492].log_data[5].valid := 1, [1492].log_data[6].valid := 1, [1492].log_data[7].valid := 1, [1492].log_data[8].valid := 1, [1492].log_data[9].valid := 1, [1492].log_data[10].valid := 1, [1492].log_data[11].valid := 1, [1492].log_data[12].valid := 1, [1492].log_data[13].valid := 1, [1492].log_data[14].valid := 1, [1492].log_data[15].valid := 1, [1492].log_data[16].valid := 1, [1492].log_data[17].valid := 1, [1492].log_data[18].valid := 1, [1492].log_data[19].valid := 1,
        [1492].time.Year := 2023, [1492].time.Month := 1, [1492].time.Day := 14, [1492].time.Hour := 20, [1492].time.Minute := 44, [1492].time.Second := 59, [1493].log_data[0].min := 1.0, [1493].log_data[0].max := 1.0, [1493].log_data[0].total := 300.0, [1493].log_data[0].time := 300.0, [1493].log_data[0].minminute := 45, [1493].log_data[0].maxminute := 45, [1493].log_data[0].valid := 1, [1493].log_data[1].valid := 1, [1493].log_data[2].valid := 1, [1493].log_data[3].valid := 1, [1493].log_data[4].valid := 1, [1493].log_data[5].valid := 1, [1493].log_data[6].valid := 1, [1493].log_data[7].valid := 1, [1493].log_data[8].valid := 1, [1493].log_data[9].valid := 1, [1493].log_data[10].valid := 1, [1493].log_data[11].valid := 1, [1493].log_data[12].valid := 1, [1493].log_data[13].valid := 1, [1493].log_data[14].valid := 1, [1493].log_data[15].valid := 1, [1493].log_data[16].valid := 1, [1493].log_data[17].valid := 1, [1493].log_data[18].valid := 1, [1493].log_data[19].valid := 1, [1493].time.Year := 2023, [1493].time.Month := 1, [1493].time.Day := 14, [1493].time.Hour := 20, [1493].time.Minute := 49, [1493].time.Second := 59, [1494].log_data[0].min := 1.0, [1494].log_data[0].max := 1.0, [1494].log_data[0].total := 300.0, [1494].log_data[0].time := 300.0, [1494].log_data[0].minminute := 50, [1494].log_data[0].maxminute := 50, [1494].log_data[0].valid := 1, [1494].log_data[1].valid := 1, [1494].log_data[2].valid := 1, [1494].log_data[3].valid := 1, [1494].log_data[4].valid := 1, [1494].log_data[5].valid := 1, [1494].log_data[6].valid := 1, [1494].log_data[7].valid := 1, [1494].log_data[8].valid := 1, [1494].log_data[9].valid := 1, [1494].log_data[10].valid := 1, [1494].log_data[11].valid := 1, [1494].log_data[12].valid := 1, [1494].log_data[13].valid := 1, [1494].log_data[14].valid := 1, [1494].log_data[15].valid := 1,
        [1494].log_data[16].valid := 1, [1494].log_data[17].valid := 1, [1494].log_data[18].valid := 1, [1494].log_data[19].valid := 1, [1494].time.Year := 2023, [1494].time.Month := 1, [1494].time.Day := 14, [1494].time.Hour := 20, [1494].time.Minute := 54, [1494].time.Second := 59, [1495].log_data[0].min := 1.0, [1495].log_data[0].max := 1.0, [1495].log_data[0].total := 300.0, [1495].log_data[0].time := 300.0, [1495].log_data[0].minminute := 55, [1495].log_data[0].maxminute := 55, [1495].log_data[0].valid := 1, [1495].log_data[1].valid := 1, [1495].log_data[2].valid := 1, [1495].log_data[3].valid := 1, [1495].log_data[4].valid := 1, [1495].log_data[5].valid := 1, [1495].log_data[6].valid := 1, [1495].log_data[7].valid := 1, [1495].log_data[8].valid := 1, [1495].log_data[9].valid := 1, [1495].log_data[10].valid := 1, [1495].log_data[11].valid := 1, [1495].log_data[12].valid := 1, [1495].log_data[13].valid := 1, [1495].log_data[14].valid := 1, [1495].log_data[15].valid := 1, [1495].log_data[16].valid := 1, [1495].log_data[17].valid := 1, [1495].log_data[18].valid := 1, [1495].log_data[19].valid := 1, [1495].time.Year := 2023, [1495].time.Month := 1, [1495].time.Day := 14, [1495].time.Hour := 20, [1495].time.Minute := 59, [1495].time.Second := 59, [1496].log_data[0].min := 1.0, [1496].log_data[0].max := 1.0, [1496].log_data[0].total := 300.0, [1496].log_data[0].time := 300.0, [1496].log_data[0].valid := 1, [1496].log_data[1].valid := 1, [1496].log_data[2].valid := 1, [1496].log_data[3].valid := 1, [1496].log_data[4].valid := 1, [1496].log_data[5].valid := 1, [1496].log_data[6].valid := 1, [1496].log_data[7].valid := 1, [1496].log_data[8].valid := 1, [1496].log_data[9].valid := 1, [1496].log_data[10].valid := 1, [1496].log_data[11].valid := 1, [1496].log_data[12].valid := 1, [1496].log_data[13].valid := 1,
        [1496].log_data[14].valid := 1, [1496].log_data[15].valid := 1, [1496].log_data[16].valid := 1, [1496].log_data[17].valid := 1, [1496].log_data[18].valid := 1, [1496].log_data[19].valid := 1, [1496].time.Year := 2023, [1496].time.Month := 1, [1496].time.Day := 14, [1496].time.Hour := 21, [1496].time.Minute := 4, [1496].time.Second := 59, [1497].log_data[0].min := 1.0, [1497].log_data[0].max := 1.0, [1497].log_data[0].total := 300.0, [1497].log_data[0].time := 300.0, [1497].log_data[0].minminute := 5, [1497].log_data[0].maxminute := 5, [1497].log_data[0].valid := 1, [1497].log_data[1].valid := 1, [1497].log_data[2].valid := 1, [1497].log_data[3].valid := 1, [1497].log_data[4].valid := 1, [1497].log_data[5].valid := 1, [1497].log_data[6].valid := 1, [1497].log_data[7].valid := 1, [1497].log_data[8].valid := 1, [1497].log_data[9].valid := 1, [1497].log_data[10].valid := 1, [1497].log_data[11].valid := 1, [1497].log_data[12].valid := 1, [1497].log_data[13].valid := 1, [1497].log_data[14].valid := 1, [1497].log_data[15].valid := 1, [1497].log_data[16].valid := 1, [1497].log_data[17].valid := 1, [1497].log_data[18].valid := 1, [1497].log_data[19].valid := 1, [1497].time.Year := 2023, [1497].time.Month := 1, [1497].time.Day := 14, [1497].time.Hour := 21, [1497].time.Minute := 9, [1497].time.Second := 59, [1498].log_data[0].min := 1.0, [1498].log_data[0].max := 1.0, [1498].log_data[0].total := 300.0, [1498].log_data[0].time := 300.0, [1498].log_data[0].minminute := 10, [1498].log_data[0].maxminute := 10, [1498].log_data[0].valid := 1, [1498].log_data[1].valid := 1, [1498].log_data[2].valid := 1, [1498].log_data[3].valid := 1, [1498].log_data[4].valid := 1, [1498].log_data[5].valid := 1, [1498].log_data[6].valid := 1, [1498].log_data[7].valid := 1, [1498].log_data[8].valid := 1, [1498].log_data[9].valid := 1,
        [1498].log_data[10].valid := 1, [1498].log_data[11].valid := 1, [1498].log_data[12].valid := 1, [1498].log_data[13].valid := 1, [1498].log_data[14].valid := 1, [1498].log_data[15].valid := 1, [1498].log_data[16].valid := 1, [1498].log_data[17].valid := 1, [1498].log_data[18].valid := 1, [1498].log_data[19].valid := 1, [1498].time.Year := 2023, [1498].time.Month := 1, [1498].time.Day := 14, [1498].time.Hour := 21, [1498].time.Minute := 14, [1498].time.Second := 59, [1499].log_data[0].min := 1.0, [1499].log_data[0].max := 1.0, [1499].log_data[0].total := 300.0, [1499].log_data[0].time := 300.0, [1499].log_data[0].minminute := 15, [1499].log_data[0].maxminute := 15, [1499].log_data[0].valid := 1, [1499].log_data[1].valid := 1, [1499].log_data[2].valid := 1, [1499].log_data[3].valid := 1, [1499].log_data[4].valid := 1, [1499].log_data[5].valid := 1, [1499].log_data[6].valid := 1, [1499].log_data[7].valid := 1, [1499].log_data[8].valid := 1, [1499].log_data[9].valid := 1, [1499].log_data[10].valid := 1, [1499].log_data[11].valid := 1, [1499].log_data[12].valid := 1, [1499].log_data[13].valid := 1, [1499].log_data[14].valid := 1, [1499].log_data[15].valid := 1, [1499].log_data[16].valid := 1, [1499].log_data[17].valid := 1, [1499].log_data[18].valid := 1, [1499].log_data[19].valid := 1, [1499].time.Year := 2023, [1499].time.Month := 1, [1499].time.Day := 14, [1499].time.Hour := 21, [1499].time.Minute := 19, [1499].time.Second := 59, [1500].log_data[0].min := 1.0, [1500].log_data[0].max := 1.0, [1500].log_data[0].total := 300.0, [1500].log_data[0].time := 300.0, [1500].log_data[0].minminute := 20, [1500].log_data[0].maxminute := 20, [1500].log_data[0].valid := 1, [1500].log_data[1].valid := 1, [1500].log_data[2].valid := 1, [1500].log_data[3].valid := 1, [1500].log_data[4].valid := 1, [1500].log_data[5].valid := 1,
        [1500].log_data[6].valid := 1, [1500].log_data[7].valid := 1, [1500].log_data[8].valid := 1, [1500].log_data[9].valid := 1, [1500].log_data[10].valid := 1, [1500].log_data[11].valid := 1, [1500].log_data[12].valid := 1, [1500].log_data[13].valid := 1, [1500].log_data[14].valid := 1, [1500].log_data[15].valid := 1, [1500].log_data[16].valid := 1, [1500].log_data[17].valid := 1, [1500].log_data[18].valid := 1, [1500].log_data[19].valid := 1, [1500].time.Year := 2023, [1500].time.Month := 1, [1500].time.Day := 14, [1500].time.Hour := 21, [1500].time.Minute := 24, [1500].time.Second := 59, [1501].log_data[0].min := 1.0, [1501].log_data[0].max := 1.0, [1501].log_data[0].total := 300.0, [1501].log_data[0].time := 300.0, [1501].log_data[0].minminute := 25, [1501].log_data[0].maxminute := 25, [1501].log_data[0].valid := 1, [1501].log_data[1].valid := 1, [1501].log_data[2].valid := 1, [1501].log_data[3].valid := 1, [1501].log_data[4].valid := 1, [1501].log_data[5].valid := 1, [1501].log_data[6].valid := 1, [1501].log_data[7].valid := 1, [1501].log_data[8].valid := 1, [1501].log_data[9].valid := 1, [1501].log_data[10].valid := 1, [1501].log_data[11].valid := 1, [1501].log_data[12].valid := 1, [1501].log_data[13].valid := 1, [1501].log_data[14].valid := 1, [1501].log_data[15].valid := 1, [1501].log_data[16].valid := 1, [1501].log_data[17].valid := 1, [1501].log_data[18].valid := 1, [1501].log_data[19].valid := 1, [1501].time.Year := 2023, [1501].time.Month := 1, [1501].time.Day := 14, [1501].time.Hour := 21, [1501].time.Minute := 29, [1501].time.Second := 59, [1502].log_data[0].min := 1.0, [1502].log_data[0].max := 1.0, [1502].log_data[0].total := 300.0, [1502].log_data[0].time := 300.0, [1502].log_data[0].minminute := 30, [1502].log_data[0].maxminute := 30, [1502].log_data[0].valid := 1, [1502].log_data[1].valid := 1,
        [1502].log_data[2].valid := 1, [1502].log_data[3].valid := 1, [1502].log_data[4].valid := 1, [1502].log_data[5].valid := 1, [1502].log_data[6].valid := 1, [1502].log_data[7].valid := 1, [1502].log_data[8].valid := 1, [1502].log_data[9].valid := 1, [1502].log_data[10].valid := 1, [1502].log_data[11].valid := 1, [1502].log_data[12].valid := 1, [1502].log_data[13].valid := 1, [1502].log_data[14].valid := 1, [1502].log_data[15].valid := 1, [1502].log_data[16].valid := 1, [1502].log_data[17].valid := 1, [1502].log_data[18].valid := 1, [1502].log_data[19].valid := 1, [1502].time.Year := 2023, [1502].time.Month := 1, [1502].time.Day := 14, [1502].time.Hour := 21, [1502].time.Minute := 34, [1502].time.Second := 59, [1503].log_data[0].min := 1.0, [1503].log_data[0].max := 1.0, [1503].log_data[0].total := 300.0, [1503].log_data[0].time := 300.0, [1503].log_data[0].minminute := 35, [1503].log_data[0].maxminute := 35, [1503].log_data[0].valid := 1, [1503].log_data[1].valid := 1, [1503].log_data[2].valid := 1, [1503].log_data[3].valid := 1, [1503].log_data[4].valid := 1, [1503].log_data[5].valid := 1, [1503].log_data[6].valid := 1, [1503].log_data[7].valid := 1, [1503].log_data[8].valid := 1, [1503].log_data[9].valid := 1, [1503].log_data[10].valid := 1, [1503].log_data[11].valid := 1, [1503].log_data[12].valid := 1, [1503].log_data[13].valid := 1, [1503].log_data[14].valid := 1, [1503].log_data[15].valid := 1, [1503].log_data[16].valid := 1, [1503].log_data[17].valid := 1, [1503].log_data[18].valid := 1, [1503].log_data[19].valid := 1, [1503].time.Year := 2023, [1503].time.Month := 1, [1503].time.Day := 14, [1503].time.Hour := 21, [1503].time.Minute := 39, [1503].time.Second := 59, [1504].log_data[0].min := 1.0, [1504].log_data[0].max := 1.0, [1504].log_data[0].total := 300.0, [1504].log_data[0].time := 300.0,
